LIN {X 0,Y 573.262,Z 487.391,A -85,B 0,C 180,E1 -2001.147,E2 -2001.147} C_VEL
LIN {X 0,Y 573.234,Z 487.393,A -85,B 0,C 180,E1 -2003.866,E2 -2003.866} C_VEL
LIN {X 0,Y 573.24,Z 487.393,A -85,B 0,C 180,E1 -2006.493,E2 -2006.493} C_VEL
LIN {X 0,Y 573.269,Z 487.389,A -85,B 0,C 180,E1 -2009.366,E2 -2009.366} C_VEL
LIN {X 0,Y 573.254,Z 487.391,A -85,B 0,C 180,E1 -2012.228,E2 -2012.228} C_VEL
LIN {X 0,Y 573.245,Z 487.394,A -85,B 0,C 180,E1 -2014.772,E2 -2014.772} C_VEL
LIN {X 0,Y 573.257,Z 487.391,A -85,B 0,C 180,E1 -2017.166,E2 -2017.166} C_VEL
LIN {X 0,Y 573.251,Z 487.39,A -85,B 0,C 180,E1 -2019.607,E2 -2019.607} C_VEL
LIN {X 0,Y 573.244,Z 487.391,A -85,B 0,C 180,E1 -2022.642,E2 -2022.642} C_VEL
LIN {X 0,Y 573.243,Z 487.392,A -85,B 0,C 180,E1 -2025.667,E2 -2025.667} C_VEL
LIN {X 0,Y 573.245,Z 487.392,A -85,B 0,C 180,E1 -2028.544,E2 -2028.544} C_VEL
LIN {X 0,Y 573.25,Z 487.391,A -85,B 0,C 180,E1 -2031.299,E2 -2031.299} C_VEL
LIN {X 0,Y 573.218,Z 487.395,A -85,B 0,C 180,E1 -2034.018,E2 -2034.018} C_VEL
LIN {X 0,Y 573.275,Z 487.389,A -85,B 0,C 180,E1 -2036.518,E2 -2036.518} C_VEL
LIN {X 0,Y 573.235,Z 487.396,A -85,B 0,C 180,E1 -2039.118,E2 -2039.118} C_VEL
LIN {X 0,Y 573.256,Z 487.393,A -85,B 0,C 180,E1 -2041.971,E2 -2041.971} C_VEL
LIN {X 0,Y 573.26,Z 487.394,A -85,B 0,C 180,E1 -2044.59,E2 -2044.59} C_VEL
LIN {X 0,Y 573.269,Z 487.559,A -85,B 0,C 180,E1 -2046.04,E2 -2046.04} C_VEL
LIN {X 0,Y 573.243,Z 493.535,A -85,B 0,C 180,E1 -2049.173,E2 -2049.173} C_VEL
LIN {X 0,Y 573.218,Z 499.051,A -85,B 0,C 180,E1 -2052.15,E2 -2052.15} C_VEL
LIN {X 0,Y 573.185,Z 504.475,A -85,B 0,C 180,E1 -2055.078,E2 -2055.078} C_VEL
LIN {X 0,Y 573.138,Z 509.987,A -85,B 0,C 180,E1 -2057.967,E2 -2057.967} C_VEL
LIN {X 0,Y 573.109,Z 515.58,A -85,B 0,C 180,E1 -2060.826,E2 -2060.826} C_VEL
LIN {X 0,Y 573.103,Z 521.654,A -85,B 0,C 180,E1 -2063.862,E2 -2063.862} C_VEL
LIN {X 0,Y 575.503,Z 530.402,A -85,B 0,C 180,E1 -2064.085,E2 -2064.085} C_VEL
LIN {X 0,Y 575.411,Z 546.369,A -85,B 0,C 180,E1 -2064.392,E2 -2064.392} C_VEL
LIN {X 0,Y 575.192,Z 562.192,A -85,B 0,C 180,E1 -2064.829,E2 -2064.829} C_VEL
LIN {X 0,Y 574.934,Z 579.816,A -85,B 0,C 180,E1 -2065.486,E2 -2065.486} C_VEL
LIN {X 0,Y 574.704,Z 595.268,A -85,B 0,C 180,E1 -2066.231,E2 -2066.231} C_VEL
LIN {X 0,Y 574.427,Z 610.317,A -85,B 0,C 180,E1 -2067.106,E2 -2067.106} C_VEL
LIN {X 0,Y 574.123,Z 625.23,A -85,B 0,C 180,E1 -2068.158,E2 -2068.158} C_VEL
LIN {X 0,Y 573.909,Z 636.875,A -85,B 0,C 180,E1 -2069.122,E2 -2069.122} C_VEL
LIN {X 0,Y 573.659,Z 649.57,A -85,B 0,C 180,E1 -2070.35,E2 -2070.35} C_VEL
LIN {X 0,Y 573.432,Z 661.888,A -85,B 0,C 180,E1 -2071.755,E2 -2071.755} C_VEL
LIN {X 0,Y 573.288,Z 672.217,A -85,B 0,C 180,E1 -2073.162,E2 -2073.162} C_VEL
LIN {X 0,Y 573.154,Z 680.969,A -85,B 0,C 180,E1 -2074.571,E2 -2074.571} C_VEL
LIN {X 0,Y 573.114,Z 688.382,A -85,B 0,C 180,E1 -2075.982,E2 -2075.982} C_VEL
LIN {X 0,Y 573.045,Z 694.49,A -85,B 0,C 180,E1 -2077.398,E2 -2077.398} C_VEL
LIN {X 0,Y 572.999,Z 699.458,A -85,B 0,C 180,E1 -2078.818,E2 -2078.818} C_VEL
LIN {X 0,Y 572.983,Z 704.181,A -85,B 0,C 180,E1 -2080.601,E2 -2080.601} C_VEL
LIN {X 0,Y 572.944,Z 706.767,A -85,B 0,C 180,E1 -2082.035,E2 -2082.035} C_VEL
LIN {X 0,Y 572.964,Z 708.381,A -85,B 0,C 180,E1 -2083.476,E2 -2083.476} C_VEL
LIN {X 0,Y 572.898,Z 708.98,A -85,B 0,C 180,E1 -2084.928,E2 -2084.928} C_VEL
LIN {X 0,Y 572.924,Z 708.532,A -85,B 0,C 180,E1 -2086.387,E2 -2086.387} C_VEL
LIN {X 0,Y 572.941,Z 707.077,A -85,B 0,C 180,E1 -2087.857,E2 -2087.857} C_VEL
LIN {X 0,Y 572.949,Z 704.49,A -85,B 0,C 180,E1 -2089.34,E2 -2089.34} C_VEL
LIN {X 0,Y 572.987,Z 700.765,A -85,B 0,C 180,E1 -2090.835,E2 -2090.835} C_VEL
LIN {X 0,Y 573.004,Z 695.804,A -85,B 0,C 180,E1 -2092.346,E2 -2092.346} C_VEL
LIN {X 0,Y 573.079,Z 689.462,A -85,B 0,C 180,E1 -2093.871,E2 -2093.871} C_VEL
LIN {X 0,Y 573.146,Z 681.566,A -85,B 0,C 180,E1 -2095.414,E2 -2095.414} C_VEL
LIN {X 0,Y 573.244,Z 673.765,A -85,B 0,C 180,E1 -2096.698,E2 -2096.698} C_VEL
LIN {X 0,Y 573.381,Z 664.059,A -85,B 0,C 180,E1 -2098.052,E2 -2098.052} C_VEL
LIN {X 0,Y 573.575,Z 653.23,A -85,B 0,C 180,E1 -2099.347,E2 -2099.347} C_VEL
LIN {X 0,Y 573.859,Z 640.374,A -85,B 0,C 180,E1 -2100.648,E2 -2100.648} C_VEL
LIN {X 0,Y 574.064,Z 627.395,A -85,B 0,C 180,E1 -2101.763,E2 -2101.763} C_VEL
LIN {X 0,Y 574.346,Z 613.444,A -85,B 0,C 180,E1 -2102.782,E2 -2102.782} C_VEL
LIN {X 0,Y 574.63,Z 597.773,A -85,B 0,C 180,E1 -2103.728,E2 -2103.728} C_VEL
LIN {X 0,Y 574.874,Z 583.699,A -85,B 0,C 180,E1 -2104.43,E2 -2104.43} C_VEL
LIN {X 0,Y 575.109,Z 568.288,A -85,B 0,C 180,E1 -2105.053,E2 -2105.053} C_VEL
LIN {X 0,Y 575.366,Z 551.011,A -85,B 0,C 180,E1 -2105.584,E2 -2105.584} C_VEL
LIN {X 0,Y 575.527,Z 534.59,A -85,B 0,C 180,E1 -2105.936,E2 -2105.936} C_VEL
LIN {X 0,Y 575.398,Z 530.006,A -85,B 0,C 180,E1 -2106.015,E2 -2106.015} C_VEL
LIN {X 0,Y 573.07,Z 521.633,A -85,B 0,C 180,E1 -2106.24,E2 -2106.24} C_VEL
LIN {X 0,Y 573.071,Z 516.673,A -85,B 0,C 180,E1 -2108.714,E2 -2108.714} C_VEL
LIN {X 0,Y 573.119,Z 511.04,A -85,B 0,C 180,E1 -2111.58,E2 -2111.58} C_VEL
LIN {X 0,Y 573.168,Z 505.123,A -85,B 0,C 180,E1 -2114.669,E2 -2114.669} C_VEL
LIN {X 0,Y 573.2,Z 500.111,A -85,B 0,C 180,E1 -2117.361,E2 -2117.361} C_VEL
LIN {X 0,Y 573.222,Z 494.449,A -85,B 0,C 180,E1 -2120.39,E2 -2120.39} C_VEL
LIN {X 0,Y 573.209,Z 489.4,A -85,B 0,C 180,E1 -2123.074,E2 -2123.074} C_VEL
LIN {X 0,Y 573.254,Z 487.395,A -85,B 0,C 180,E1 -2124.076,E2 -2124.076} C_VEL
LIN {X 0,Y 573.278,Z 487.391,A -85,B 0,C 180,E1 -2126.518,E2 -2126.518} C_VEL
LIN {X 0,Y 573.237,Z 487.395,A -85,B 0,C 180,E1 -2129.114,E2 -2129.114} C_VEL
LIN {X 0,Y 573.257,Z 487.393,A -85,B 0,C 180,E1 -2131.967,E2 -2131.967} C_VEL
LIN {X 0,Y 573.252,Z 487.393,A -85,B 0,C 180,E1 -2134.589,E2 -2134.589} C_VEL
LIN {X 0,Y 573.255,Z 487.39,A -85,B 0,C 180,E1 -2136.901,E2 -2136.901} C_VEL
LIN {X 0,Y 573.247,Z 487.392,A -85,B 0,C 180,E1 -2139.923,E2 -2139.923} C_VEL
LIN {X 0,Y 573.255,Z 487.395,A -85,B 0,C 180,E1 -2142.987,E2 -2142.987} C_VEL
LIN {X 0,Y 573.264,Z 487.392,A -85,B 0,C 180,E1 -2145.806,E2 -2145.806} C_VEL
LIN {X 0,Y 573.273,Z 487.389,A -85,B 0,C 180,E1 -2148.733,E2 -2148.733} C_VEL
LIN {X 0,Y 573.3,Z 487.385,A -85,B 0,C 180,E1 -2151.54,E2 -2151.54} C_VEL
LIN {X 0,Y 573.295,Z 487.385,A -85,B 0,C 180,E1 -2154.372,E2 -2154.372} C_VEL
LIN {X 0,Y 573.31,Z 487.387,A -85,B 0,C 180,E1 -2157.892,E2 -2157.892} C_VEL
LIN {X 0,Y 573.331,Z 487.385,A -85,B 0,C 180,E1 -2160.702,E2 -2160.702} C_VEL
LIN {X 0,Y 573.234,Z 487.396,A -85,B 0,C 180,E1 -2163.514,E2 -2163.514} C_VEL
LIN {X 0,Y 573.284,Z 487.385,A -85,B 0,C 180,E1 -2165.628,E2 -2165.628} C_VEL
LIN {X 0,Y 573.298,Z 487.385,A -85,B 0,C 180,E1 -2168.459,E2 -2168.459} C_VEL
LIN {X 0,Y 573.288,Z 487.388,A -85,B 0,C 180,E1 -2171.311,E2 -2171.311} C_VEL
LIN {X 0,Y 573.27,Z 487.391,A -85,B 0,C 180,E1 -2174.425,E2 -2174.425} C_VEL
LIN {X 0,Y 573.249,Z 487.387,A -85,B 0,C 180,E1 -2177.112,E2 -2177.112} C_VEL
LIN {X 0,Y 573.248,Z 487.392,A -85,B 0,C 180,E1 -2180.076,E2 -2180.076} C_VEL
LIN {X 0,Y 573.261,Z 487.388,A -85,B 0,C 180,E1 -2183.154,E2 -2183.154} C_VEL
LIN {X 0,Y 573.281,Z 487.386,A -85,B 0,C 180,E1 -2186.189,E2 -2186.189} C_VEL
LIN {X 0,Y 573.234,Z 487.393,A -85,B 0,C 180,E1 -2188.564,E2 -2188.564} C_VEL
LIN {X 0,Y 573.231,Z 487.394,A -85,B 0,C 180,E1 -2190.993,E2 -2190.993} C_VEL
LIN {X 0,Y 573.278,Z 487.389,A -85,B 0,C 180,E1 -2193.529,E2 -2193.529} C_VEL
LIN {X 0,Y 573.253,Z 487.394,A -85,B 0,C 180,E1 -2196.048,E2 -2196.048} C_VEL
LIN {X 0,Y 573.241,Z 487.396,A -85,B 0,C 180,E1 -2198.701,E2 -2198.701} C_VEL
LIN {X 0,Y 573.257,Z 487.393,A -85,B 0,C 180,E1 -2201.598,E2 -2201.598} C_VEL
LIN {X 0,Y 573.23,Z 487.397,A -85,B 0,C 180,E1 -2204.334,E2 -2204.334} C_VEL
LIN {X 0,Y 573.253,Z 487.393,A -85,B 0,C 180,E1 -2207.357,E2 -2207.357} C_VEL
LIN {X 0,Y 573.267,Z 487.459,A -85,B 0,C 180,E1 -2208.403,E2 -2208.403} C_VEL
LIN {X 0,Y 574.646,Z 493.703,A -85,B 0,C 180,E1 -2210.046,E2 -2210.046} C_VEL
LIN {X 0,Y 574.7,Z 501.177,A -85,B 0,C 180,E1 -2211.906,E2 -2211.906} C_VEL
LIN {X 0,Y 574.476,Z 511.898,A -85,B 0,C 180,E1 -2214.473,E2 -2214.473} C_VEL
LIN {X 0,Y 574.26,Z 522.796,A -85,B 0,C 180,E1 -2217.004,E2 -2217.004} C_VEL
LIN {X 0,Y 574.097,Z 535.51,A -85,B 0,C 180,E1 -2219.874,E2 -2219.874} C_VEL
LIN {X 0,Y 573.926,Z 548.224,A -85,B 0,C 180,E1 -2222.665,E2 -2222.665} C_VEL
LIN {X 0,Y 573.714,Z 560.938,A -85,B 0,C 180,E1 -2225.387,E2 -2225.387} C_VEL
LIN {X 0,Y 573.592,Z 573.652,A -85,B 0,C 180,E1 -2228.057,E2 -2228.057} C_VEL
LIN {X 0,Y 573.576,Z 577.286,A -85,B 0,C 180,E1 -2228.785,E2 -2228.785} C_VEL
LIN {X 0,Y 575.538,Z 585.817,A -85,B 0,C 180,E1 -2228.972,E2 -2228.972} C_VEL
LIN {X 0,Y 575.425,Z 602.393,A -85,B 0,C 180,E1 -2229.257,E2 -2229.257} C_VEL
LIN {X 0,Y 575.273,Z 618.484,A -85,B 0,C 180,E1 -2229.672,E2 -2229.672} C_VEL
LIN {X 0,Y 575.028,Z 635.073,A -85,B 0,C 180,E1 -2230.249,E2 -2230.249} C_VEL
LIN {X 0,Y 574.764,Z 650.013,A -85,B 0,C 180,E1 -2230.909,E2 -2230.909} C_VEL
LIN {X 0,Y 574.509,Z 665.029,A -85,B 0,C 180,E1 -2231.732,E2 -2231.732} C_VEL
LIN {X 0,Y 574.21,Z 679.457,A -85,B 0,C 180,E1 -2232.682,E2 -2232.682} C_VEL
LIN {X 0,Y 573.971,Z 692.926,A -85,B 0,C 180,E1 -2233.735,E2 -2233.735} C_VEL
LIN {X 0,Y 573.729,Z 705.738,A -85,B 0,C 180,E1 -2234.913,E2 -2234.913} C_VEL
LIN {X 0,Y 573.511,Z 717.451,A -85,B 0,C 180,E1 -2236.176,E2 -2236.176} C_VEL
LIN {X 0,Y 573.33,Z 728.738,A -85,B 0,C 180,E1 -2237.614,E2 -2237.614} C_VEL
LIN {X 0,Y 573.204,Z 738.357,A -85,B 0,C 180,E1 -2239.074,E2 -2239.074} C_VEL
LIN {X 0,Y 573.109,Z 746.053,A -85,B 0,C 180,E1 -2240.472,E2 -2240.472} C_VEL
LIN {X 0,Y 573.054,Z 752.628,A -85,B 0,C 180,E1 -2241.893,E2 -2241.893} C_VEL
LIN {X 0,Y 573.025,Z 758.391,A -85,B 0,C 180,E1 -2243.433,E2 -2243.433} C_VEL
LIN {X 0,Y 573.035,Z 761.249,A -85,B 0,C 180,E1 -2244.37,E2 -2244.37} C_VEL
LIN {X 0,Y 573.006,Z 764.636,A -85,B 0,C 180,E1 -2245.781,E2 -2245.781} C_VEL
LIN {X 0,Y 572.947,Z 767.089,A -85,B 0,C 180,E1 -2247.188,E2 -2247.188} C_VEL
LIN {X 0,Y 572.943,Z 768.479,A -85,B 0,C 180,E1 -2248.595,E2 -2248.595} C_VEL
LIN {X 0,Y 572.933,Z 769,A -85,B 0,C 180,E1 -2250.001,E2 -2250.001} C_VEL
LIN {X 0,Y 572.943,Z 768.478,A -85,B 0,C 180,E1 -2251.407,E2 -2251.407} C_VEL
LIN {X 0,Y 572.947,Z 767.086,A -85,B 0,C 180,E1 -2252.813,E2 -2252.813} C_VEL
LIN {X 0,Y 573.006,Z 764.633,A -85,B 0,C 180,E1 -2254.221,E2 -2254.221} C_VEL
LIN {X 0,Y 573.012,Z 760.184,A -85,B 0,C 180,E1 -2255.985,E2 -2255.985} C_VEL
LIN {X 0,Y 573.043,Z 755.466,A -85,B 0,C 180,E1 -2257.4,E2 -2257.4} C_VEL
LIN {X 0,Y 573.092,Z 747.854,A -85,B 0,C 180,E1 -2259.174,E2 -2259.174} C_VEL
LIN {X 0,Y 573.15,Z 740.257,A -85,B 0,C 180,E1 -2260.599,E2 -2260.599} C_VEL
LIN {X 0,Y 573.304,Z 731.205,A -85,B 0,C 180,E1 -2262.029,E2 -2262.029} C_VEL
LIN {X 0,Y 573.442,Z 720.418,A -85,B 0,C 180,E1 -2263.466,E2 -2263.466} C_VEL
LIN {X 0,Y 573.658,Z 709.292,A -85,B 0,C 180,E1 -2264.726,E2 -2264.726} C_VEL
LIN {X 0,Y 573.902,Z 697.137,A -85,B 0,C 180,E1 -2265.903,E2 -2265.903} C_VEL
LIN {X 0,Y 574.132,Z 683.875,A -85,B 0,C 180,E1 -2266.994,E2 -2266.994} C_VEL
LIN {X 0,Y 574.431,Z 669.425,A -85,B 0,C 180,E1 -2267.995,E2 -2267.995} C_VEL
LIN {X 0,Y 574.662,Z 655.255,A -85,B 0,C 180,E1 -2268.818,E2 -2268.818} C_VEL
LIN {X 0,Y 574.935,Z 640.706,A -85,B 0,C 180,E1 -2269.521,E2 -2269.521} C_VEL
LIN {X 0,Y 575.198,Z 624.331,A -85,B 0,C 180,E1 -2270.146,E2 -2270.146} C_VEL
LIN {X 0,Y 575.387,Z 608.329,A -85,B 0,C 180,E1 -2270.606,E2 -2270.606} C_VEL
LIN {X 0,Y 575.518,Z 591.668,A -85,B 0,C 180,E1 -2270.94,E2 -2270.94} C_VEL
LIN {X 0,Y 575.396,Z 584.289,A -85,B 0,C 180,E1 -2271.053,E2 -2271.053} C_VEL
LIN {X 0,Y 573.548,Z 577.09,A -85,B 0,C 180,E1 -2271.23,E2 -2271.23} C_VEL
LIN {X 0,Y 573.695,Z 562.746,A -85,B 0,C 180,E1 -2274.23,E2 -2274.23} C_VEL
LIN {X 0,Y 573.889,Z 550.032,A -85,B 0,C 180,E1 -2276.944,E2 -2276.944} C_VEL
LIN {X 0,Y 574.052,Z 536.852,A -85,B 0,C 180,E1 -2279.829,E2 -2279.829} C_VEL
LIN {X 0,Y 574.247,Z 524.604,A -85,B 0,C 180,E1 -2282.582,E2 -2282.582} C_VEL
LIN {X 0,Y 574.398,Z 513.707,A -85,B 0,C 180,E1 -2285.105,E2 -2285.105} C_VEL
LIN {X 0,Y 574.654,Z 502.809,A -85,B 0,C 180,E1 -2287.698,E2 -2287.698} C_VEL
LIN {X 0,Y 574.733,Z 495.035,A -85,B 0,C 180,E1 -2289.612,E2 -2289.612} C_VEL
LIN {X 0,Y 573.722,Z 489.451,A -85,B 0,C 180,E1 -2291.076,E2 -2291.076} C_VEL
LIN {X 0,Y 573.26,Z 487.39,A -85,B 0,C 180,E1 -2291.539,E2 -2291.539} C_VEL
LIN {X 0,Y 573.241,Z 487.392,A -85,B 0,C 180,E1 -2294.333,E2 -2294.333} C_VEL
LIN {X 0,Y 573.244,Z 487.389,A -85,B 0,C 180,E1 -2297.358,E2 -2297.358} C_VEL
LIN {X 0,Y 573.249,Z 487.394,A -85,B 0,C 180,E1 -2300.393,E2 -2300.393} C_VEL
LIN {X 0,Y 573.253,Z 487.388,A -85,B 0,C 180,E1 -2303.078,E2 -2303.078} C_VEL
LIN {X 0,Y 573.272,Z 487.385,A -85,B 0,C 180,E1 -2305.672,E2 -2305.672} C_VEL
LIN {X 0,Y 573.242,Z 487.396,A -85,B 0,C 180,E1 -2308.185,E2 -2308.185} C_VEL
LIN {X 0,Y 573.267,Z 487.388,A -85,B 0,C 180,E1 -2310.635,E2 -2310.635} C_VEL
LIN {X 0,Y 573.252,Z 487.387,A -85,B 0,C 180,E1 -2313.024,E2 -2313.024} C_VEL
LIN {X 0,Y 573.277,Z 487.386,A -85,B 0,C 180,E1 -2315.366,E2 -2315.366} C_VEL
LIN {X 0,Y 573.231,Z 487.393,A -85,B 0,C 180,E1 -2318.42,E2 -2318.42} C_VEL
LIN {X 0,Y 573.265,Z 487.387,A -85,B 0,C 180,E1 -2318.952,E2 -2318.952} C_VEL
LIN {X 0,Y 575.047,Z 492.214,A -85,B 0,C 180,E1 -2319.094,E2 -2319.094} C_VEL
LIN {X 0,Y 575.537,Z 494.378,A -85,B 0,C 180,E1 -2319.147,E2 -2319.147} C_VEL
LIN {X 0,Y 575.338,Z 511.225,A -85,B 0,C 180,E1 -2319.51,E2 -2319.51} C_VEL
LIN {X 0,Y 575.13,Z 527.051,A -85,B 0,C 180,E1 -2319.992,E2 -2319.992} C_VEL
LIN {X 0,Y 574.918,Z 543.212,A -85,B 0,C 180,E1 -2320.637,E2 -2320.637} C_VEL
LIN {X 0,Y 574.637,Z 557.901,A -85,B 0,C 180,E1 -2321.367,E2 -2321.367} C_VEL
LIN {X 0,Y 574.38,Z 572.82,A -85,B 0,C 180,E1 -2322.27,E2 -2322.27} C_VEL
LIN {X 0,Y 574.107,Z 586.828,A -85,B 0,C 180,E1 -2323.281,E2 -2323.281} C_VEL
LIN {X 0,Y 573.826,Z 599.609,A -85,B 0,C 180,E1 -2324.369,E2 -2324.369} C_VEL
LIN {X 0,Y 573.632,Z 611.874,A -85,B 0,C 180,E1 -2325.594,E2 -2325.594} C_VEL
LIN {X 0,Y 573.419,Z 622.99,A -85,B 0,C 180,E1 -2326.895,E2 -2326.895} C_VEL
LIN {X 0,Y 573.288,Z 633.371,A -85,B 0,C 180,E1 -2328.33,E2 -2328.33} C_VEL
LIN {X 0,Y 573.169,Z 642.045,A -85,B 0,C 180,E1 -2329.759,E2 -2329.759} C_VEL
LIN {X 0,Y 573.086,Z 649.296,A -85,B 0,C 180,E1 -2331.183,E2 -2331.183} C_VEL
LIN {X 0,Y 573.044,Z 655.298,A -85,B 0,C 180,E1 -2332.601,E2 -2332.601} C_VEL
LIN {X 0,Y 573.014,Z 660.066,A -85,B 0,C 180,E1 -2334.016,E2 -2334.016} C_VEL
LIN {X 0,Y 573.005,Z 664.546,A -85,B 0,C 180,E1 -2335.78,E2 -2335.78} C_VEL
LIN {X 0,Y 572.954,Z 667.024,A -85,B 0,C 180,E1 -2337.188,E2 -2337.188} C_VEL
LIN {X 0,Y 572.939,Z 668.459,A -85,B 0,C 180,E1 -2338.595,E2 -2338.595} C_VEL
LIN {X 0,Y 572.935,Z 668.996,A -85,B 0,C 180,E1 -2340,E2 -2340} C_VEL
LIN {X 0,Y 572.939,Z 668.518,A -85,B 0,C 180,E1 -2341.406,E2 -2341.406} C_VEL
LIN {X 0,Y 572.954,Z 667.141,A -85,B 0,C 180,E1 -2342.813,E2 -2342.813} C_VEL
LIN {X 0,Y 573.006,Z 664.733,A -85,B 0,C 180,E1 -2344.221,E2 -2344.221} C_VEL
LIN {X 0,Y 573.017,Z 660.331,A -85,B 0,C 180,E1 -2345.984,E2 -2345.984} C_VEL
LIN {X 0,Y 573.044,Z 655.624,A -85,B 0,C 180,E1 -2347.399,E2 -2347.399} C_VEL
LIN {X 0,Y 573.082,Z 649.694,A -85,B 0,C 180,E1 -2348.818,E2 -2348.818} C_VEL
LIN {X 0,Y 573.186,Z 641.542,A -85,B 0,C 180,E1 -2350.42,E2 -2350.42} C_VEL
LIN {X 0,Y 573.271,Z 632.765,A -85,B 0,C 180,E1 -2351.85,E2 -2351.85} C_VEL
LIN {X 0,Y 573.437,Z 622.274,A -85,B 0,C 180,E1 -2353.286,E2 -2353.286} C_VEL
LIN {X 0,Y 573.638,Z 610.405,A -85,B 0,C 180,E1 -2354.655,E2 -2354.655} C_VEL
LIN {X 0,Y 573.86,Z 598.613,A -85,B 0,C 180,E1 -2355.813,E2 -2355.813} C_VEL
LIN {X 0,Y 574.115,Z 585.624,A -85,B 0,C 180,E1 -2356.902,E2 -2356.902} C_VEL
LIN {X 0,Y 574.378,Z 571.555,A -85,B 0,C 180,E1 -2357.904,E2 -2357.904} C_VEL
LIN {X 0,Y 574.652,Z 557.869,A -85,B 0,C 180,E1 -2358.726,E2 -2358.726} C_VEL
LIN {X 0,Y 574.939,Z 541.855,A -85,B 0,C 180,E1 -2359.515,E2 -2359.515} C_VEL
LIN {X 0,Y 574.989,Z 538.259,A -85,B 0,C 180,E1 -2359.667,E2 -2359.667} C_VEL
LIN {X 0,Y 574.341,Z 534.687,A -85,B 0,C 180,E1 -2359.839,E2 -2359.839} C_VEL
LIN {X 0,Y 569.101,Z 523.749,A -85,B 0,C 180,E1 -2360.438,E2 -2360.438} C_VEL
LIN {X 0,Y 568.59,Z 520.064,A -85,B 0,C 180,E1 -2360.573,E2 -2360.573} C_VEL
LIN {X 0,Y 568.788,Z 505.313,A -85,B 0,C 180,E1 -2360.974,E2 -2360.974} C_VEL
LIN {X 0,Y 568.718,Z 494.777,A -85,B 0,C 180,E1 -2361.195,E2 -2361.195} C_VEL
LIN {X 0,Y 566.315,Z 488.81,A -85,B 0,C 180,E1 -2361.387,E2 -2361.387} C_VEL
LIN {X 0,Y 566.221,Z 488.269,A -85,B 0,C 180,E1 -2361.423,E2 -2361.423} C_VEL
LIN {X 0,Y 566.201,Z 488.27,A -85,B 0,C 180,E1 -2364.181,E2 -2364.181} C_VEL
LIN {X 0,Y 566.211,Z 488.268,A -85,B 0,C 180,E1 -2366.659,E2 -2366.659} C_VEL
LIN {X 0,Y 566.196,Z 488.274,A -85,B 0,C 180,E1 -2368.954,E2 -2368.954} C_VEL
LIN {X 0,Y 566.196,Z 488.271,A -85,B 0,C 180,E1 -2371.422,E2 -2371.422} C_VEL
LIN {X 0,Y 566.215,Z 488.267,A -85,B 0,C 180,E1 -2373.956,E2 -2373.956} C_VEL
LIN {X 0,Y 566.219,Z 488.266,A -85,B 0,C 180,E1 -2376.569,E2 -2376.569} C_VEL
LIN {X 0,Y 566.226,Z 488.265,A -85,B 0,C 180,E1 -2379.687,E2 -2379.687} C_VEL
LIN {X 0,Y 566.206,Z 488.27,A -85,B 0,C 180,E1 -2382.917,E2 -2382.917} C_VEL
LIN {X 0,Y 566.207,Z 488.273,A -85,B 0,C 180,E1 -2386.048,E2 -2386.048} C_VEL
LIN {X 0,Y 566.214,Z 488.271,A -85,B 0,C 180,E1 -2388.864,E2 -2388.864} C_VEL
LIN {X 0,Y 566.192,Z 488.273,A -85,B 0,C 180,E1 -2391.637,E2 -2391.637} C_VEL
LIN {X 0,Y 566.168,Z 488.275,A -85,B 0,C 180,E1 -2394.308,E2 -2394.308} C_VEL
LIN {X 0,Y 566.226,Z 488.266,A -85,B 0,C 180,E1 -2396.898,E2 -2396.898} C_VEL
LIN {X 0,Y 566.187,Z 488.272,A -85,B 0,C 180,E1 -2399.407,E2 -2399.407} C_VEL
LIN {X 0,Y 566.218,Z 488.271,A -85,B 0,C 180,E1 -2401.857,E2 -2401.857} C_VEL
LIN {X 0,Y 566.22,Z 488.268,A -85,B 0,C 180,E1 -2404.251,E2 -2404.251} C_VEL
LIN {X 0,Y 566.233,Z 488.393,A -85,B 0,C 180,E1 -2406.015,E2 -2406.015} C_VEL
LIN {X 0,Y 566.204,Z 493.917,A -85,B 0,C 180,E1 -2408.902,E2 -2408.902} C_VEL
LIN {X 0,Y 566.172,Z 498.111,A -85,B 0,C 180,E1 -2411.171,E2 -2411.171} C_VEL
LIN {X 0,Y 566.115,Z 503.525,A -85,B 0,C 180,E1 -2414.15,E2 -2414.15} C_VEL
LIN {X 0,Y 566.106,Z 507.629,A -85,B 0,C 180,E1 -2416.356,E2 -2416.356} C_VEL
LIN {X 0,Y 566.061,Z 513.177,A -85,B 0,C 180,E1 -2419.266,E2 -2419.266} C_VEL
LIN {X 0,Y 566.038,Z 518.808,A -85,B 0,C 180,E1 -2422.149,E2 -2422.149} C_VEL
LIN {X 0,Y 566.046,Z 521.652,A -85,B 0,C 180,E1 -2423.583,E2 -2423.583} C_VEL
LIN {X 0,Y 568.894,Z 532.268,A -85,B 0,C 180,E1 -2423.861,E2 -2423.861} C_VEL
LIN {X 0,Y 568.745,Z 548.595,A -85,B 0,C 180,E1 -2424.193,E2 -2424.193} C_VEL
LIN {X 0,Y 568.475,Z 566.381,A -85,B 0,C 180,E1 -2424.724,E2 -2424.724} C_VEL
LIN {X 0,Y 568.181,Z 581,A -85,B 0,C 180,E1 -2425.299,E2 -2425.299} C_VEL
LIN {X 0,Y 567.92,Z 595.456,A -85,B 0,C 180,E1 -2426.008,E2 -2426.008} C_VEL
LIN {X 0,Y 567.595,Z 610.488,A -85,B 0,C 180,E1 -2426.894,E2 -2426.894} C_VEL
LIN {X 0,Y 567.255,Z 625.366,A -85,B 0,C 180,E1 -2427.958,E2 -2427.958} C_VEL
LIN {X 0,Y 566.997,Z 636.987,A -85,B 0,C 180,E1 -2428.934,E2 -2428.934} C_VEL
LIN {X 0,Y 566.688,Z 649.676,A -85,B 0,C 180,E1 -2430.177,E2 -2430.177} C_VEL
LIN {X 0,Y 566.41,Z 661.983,A -85,B 0,C 180,E1 -2431.599,E2 -2431.599} C_VEL
LIN {X 0,Y 566.251,Z 672.285,A -85,B 0,C 180,E1 -2433.023,E2 -2433.023} C_VEL
LIN {X 0,Y 566.117,Z 681.027,A -85,B 0,C 180,E1 -2434.449,E2 -2434.449} C_VEL
LIN {X 0,Y 566.029,Z 689.237,A -85,B 0,C 180,E1 -2436.057,E2 -2436.057} C_VEL
LIN {X 0,Y 565.972,Z 695.228,A -85,B 0,C 180,E1 -2437.491,E2 -2437.491} C_VEL
LIN {X 0,Y 565.895,Z 700.022,A -85,B 0,C 180,E1 -2438.93,E2 -2438.93} C_VEL
LIN {X 0,Y 565.9,Z 702.958,A -85,B 0,C 180,E1 -2440.012,E2 -2440.012} C_VEL
LIN {X 0,Y 565.873,Z 705.93,A -85,B 0,C 180,E1 -2441.461,E2 -2441.461} C_VEL
LIN {X 0,Y 565.838,Z 707.906,A -85,B 0,C 180,E1 -2442.918,E2 -2442.918} C_VEL
LIN {X 0,Y 565.84,Z 708.856,A -85,B 0,C 180,E1 -2444.382,E2 -2444.382} C_VEL
LIN {X 0,Y 565.804,Z 708.809,A -85,B 0,C 180,E1 -2445.858,E2 -2445.858} C_VEL
LIN {X 0,Y 565.83,Z 707.72,A -85,B 0,C 180,E1 -2447.342,E2 -2447.342} C_VEL
LIN {X 0,Y 565.85,Z 705.599,A -85,B 0,C 180,E1 -2448.839,E2 -2448.839} C_VEL
LIN {X 0,Y 565.89,Z 702.287,A -85,B 0,C 180,E1 -2450.348,E2 -2450.348} C_VEL
LIN {X 0,Y 565.931,Z 697.776,A -85,B 0,C 180,E1 -2451.872,E2 -2451.872} C_VEL
LIN {X 0,Y 565.977,Z 691.966,A -85,B 0,C 180,E1 -2453.412,E2 -2453.412} C_VEL
LIN {X 0,Y 566.035,Z 686.622,A -85,B 0,C 180,E1 -2454.578,E2 -2454.578} C_VEL
LIN {X 0,Y 566.174,Z 678.134,A -85,B 0,C 180,E1 -2456.145,E2 -2456.145} C_VEL
LIN {X 0,Y 566.315,Z 667.674,A -85,B 0,C 180,E1 -2457.733,E2 -2457.733} C_VEL
LIN {X 0,Y 566.485,Z 658.349,A -85,B 0,C 180,E1 -2458.936,E2 -2458.936} C_VEL
LIN {X 0,Y 566.726,Z 647.425,A -85,B 0,C 180,E1 -2460.147,E2 -2460.147} C_VEL
LIN {X 0,Y 566.995,Z 636.403,A -85,B 0,C 180,E1 -2461.21,E2 -2461.21} C_VEL
LIN {X 0,Y 567.279,Z 622.959,A -85,B 0,C 180,E1 -2462.324,E2 -2462.324} C_VEL
LIN {X 0,Y 567.63,Z 608.469,A -85,B 0,C 180,E1 -2463.326,E2 -2463.326} C_VEL
LIN {X 0,Y 567.889,Z 595.643,A -85,B 0,C 180,E1 -2464.073,E2 -2464.073} C_VEL
LIN {X 0,Y 568.171,Z 581.485,A -85,B 0,C 180,E1 -2464.769,E2 -2464.769} C_VEL
LIN {X 0,Y 568.438,Z 566.657,A -85,B 0,C 180,E1 -2465.358,E2 -2465.358} C_VEL
LIN {X 0,Y 568.699,Z 548.636,A -85,B 0,C 180,E1 -2465.898,E2 -2465.898} C_VEL
LIN {X 0,Y 568.902,Z 532.727,A -85,B 0,C 180,E1 -2466.222,E2 -2466.222} C_VEL
LIN {X 0,Y 568.39,Z 530.003,A -85,B 0,C 180,E1 -2466.286,E2 -2466.286} C_VEL
LIN {X 0,Y 565.989,Z 521.644,A -85,B 0,C 180,E1 -2466.513,E2 -2466.513} C_VEL
LIN {X 0,Y 565.999,Z 516.161,A -85,B 0,C 180,E1 -2469.29,E2 -2469.29} C_VEL
LIN {X 0,Y 566.062,Z 510.729,A -85,B 0,C 180,E1 -2472.099,E2 -2472.099} C_VEL
LIN {X 0,Y 566.126,Z 505.189,A -85,B 0,C 180,E1 -2475.039,E2 -2475.039} C_VEL
LIN {X 0,Y 566.137,Z 499.958,A -85,B 0,C 180,E1 -2477.905,E2 -2477.905} C_VEL
LIN {X 0,Y 566.172,Z 494.608,A -85,B 0,C 180,E1 -2480.722,E2 -2480.722} C_VEL
LIN {X 0,Y 566.155,Z 489.489,A -85,B 0,C 180,E1 -2483.426,E2 -2483.426} C_VEL
LIN {X 0,Y 566.204,Z 488.273,A -85,B 0,C 180,E1 -2484.048,E2 -2484.048} C_VEL
LIN {X 0,Y 566.222,Z 488.271,A -85,B 0,C 180,E1 -2486.898,E2 -2486.898} C_VEL
LIN {X 0,Y 566.187,Z 488.276,A -85,B 0,C 180,E1 -2489.407,E2 -2489.407} C_VEL
LIN {X 0,Y 566.22,Z 488.269,A -85,B 0,C 180,E1 -2491.857,E2 -2491.857} C_VEL
LIN {X 0,Y 566.22,Z 488.267,A -85,B 0,C 180,E1 -2494.251,E2 -2494.251} C_VEL
LIN {X 0,Y 566.226,Z 488.266,A -85,B 0,C 180,E1 -2496.702,E2 -2496.702} C_VEL
LIN {X 0,Y 566.21,Z 488.268,A -85,B 0,C 180,E1 -2499.662,E2 -2499.662} C_VEL
LIN {X 0,Y 566.197,Z 488.271,A -85,B 0,C 180,E1 -2502.668,E2 -2502.668} C_VEL
LIN {X 0,Y 566.225,Z 488.27,A -85,B 0,C 180,E1 -2505.626,E2 -2505.626} C_VEL
LIN {X 0,Y 566.265,Z 488.262,A -85,B 0,C 180,E1 -2508.653,E2 -2508.653} C_VEL
LIN {X 0,Y 566.242,Z 488.264,A -85,B 0,C 180,E1 -2511.434,E2 -2511.434} C_VEL
LIN {X 0,Y 566.263,Z 488.261,A -85,B 0,C 180,E1 -2514.301,E2 -2514.301} C_VEL
LIN {X 0,Y 566.28,Z 488.263,A -85,B 0,C 180,E1 -2517.866,E2 -2517.866} C_VEL
LIN {X 0,Y 566.3,Z 488.26,A -85,B 0,C 180,E1 -2520.711,E2 -2520.711} C_VEL
LIN {X 0,Y 566.271,Z 488.26,A -85,B 0,C 180,E1 -2522.845,E2 -2522.845} C_VEL
LIN {X 0,Y 566.252,Z 488.261,A -85,B 0,C 180,E1 -2525.698,E2 -2525.698} C_VEL
LIN {X 0,Y 566.239,Z 488.265,A -85,B 0,C 180,E1 -2528.565,E2 -2528.565} C_VEL
LIN {X 0,Y 566.24,Z 488.267,A -85,B 0,C 180,E1 -2531.454,E2 -2531.454} C_VEL
LIN {X 0,Y 566.223,Z 488.268,A -85,B 0,C 180,E1 -2534.507,E2 -2534.507} C_VEL
LIN {X 0,Y 566.194,Z 488.263,A -85,B 0,C 180,E1 -2537.332,E2 -2537.332} C_VEL
LIN {X 0,Y 566.21,Z 488.267,A -85,B 0,C 180,E1 -2540.337,E2 -2540.337} C_VEL
LIN {X 0,Y 566.22,Z 488.265,A -85,B 0,C 180,E1 -2543.402,E2 -2543.402} C_VEL
LIN {X 0,Y 566.218,Z 488.264,A -85,B 0,C 180,E1 -2545.748,E2 -2545.748} C_VEL
LIN {X 0,Y 566.198,Z 488.27,A -85,B 0,C 180,E1 -2548.204,E2 -2548.204} C_VEL
LIN {X 0,Y 566.185,Z 488.275,A -85,B 0,C 180,E1 -2550.592,E2 -2550.592} C_VEL
LIN {X 0,Y 566.219,Z 488.269,A -85,B 0,C 180,E1 -2553.102,E2 -2553.102} C_VEL
LIN {X 0,Y 566.204,Z 488.269,A -85,B 0,C 180,E1 -2555.689,E2 -2555.689} C_VEL
LIN {X 0,Y 566.208,Z 488.271,A -85,B 0,C 180,E1 -2558.56,E2 -2558.56} C_VEL
LIN {X 0,Y 566.213,Z 488.269,A -85,B 0,C 180,E1 -2561.136,E2 -2561.136} C_VEL
LIN {X 0,Y 566.191,Z 488.274,A -85,B 0,C 180,E1 -2564.036,E2 -2564.036} C_VEL
LIN {X 0,Y 566.206,Z 488.272,A -85,B 0,C 180,E1 -2567.082,E2 -2567.082} C_VEL
LIN {X 0,Y 566.264,Z 488.36,A -85,B 0,C 180,E1 -2568.096,E2 -2568.096} C_VEL
LIN {X 0,Y 567.902,Z 496.189,A -85,B 0,C 180,E1 -2570.109,E2 -2570.109} C_VEL
LIN {X 0,Y 567.836,Z 505.294,A -85,B 0,C 180,E1 -2572.383,E2 -2572.383} C_VEL
LIN {X 0,Y 567.563,Z 517.347,A -85,B 0,C 180,E1 -2575.279,E2 -2575.279} C_VEL
LIN {X 0,Y 567.305,Z 530.061,A -85,B 0,C 180,E1 -2578.232,E2 -2578.232} C_VEL
LIN {X 0,Y 567.06,Z 542.775,A -85,B 0,C 180,E1 -2581.096,E2 -2581.096} C_VEL
LIN {X 0,Y 566.876,Z 553.673,A -85,B 0,C 180,E1 -2583.493,E2 -2583.493} C_VEL
LIN {X 0,Y 566.694,Z 566.388,A -85,B 0,C 180,E1 -2586.232,E2 -2586.232} C_VEL
LIN {X 0,Y 566.581,Z 577.12,A -85,B 0,C 180,E1 -2588.502,E2 -2588.502} C_VEL
LIN {X 0,Y 568.936,Z 586.825,A -85,B 0,C 180,E1 -2588.73,E2 -2588.73} C_VEL
LIN {X 0,Y 568.781,Z 603.534,A -85,B 0,C 180,E1 -2589.027,E2 -2589.027} C_VEL
LIN {X 0,Y 568.583,Z 620.002,A -85,B 0,C 180,E1 -2589.469,E2 -2589.469} C_VEL
LIN {X 0,Y 568.299,Z 635.651,A -85,B 0,C 180,E1 -2590.029,E2 -2590.029} C_VEL
LIN {X 0,Y 568.027,Z 650.012,A -85,B 0,C 180,E1 -2590.673,E2 -2590.673} C_VEL
LIN {X 0,Y 567.701,Z 665.031,A -85,B 0,C 180,E1 -2591.505,E2 -2591.505} C_VEL
LIN {X 0,Y 567.386,Z 679.14,A -85,B 0,C 180,E1 -2592.444,E2 -2592.444} C_VEL
LIN {X 0,Y 567.087,Z 692.927,A -85,B 0,C 180,E1 -2593.532,E2 -2593.532} C_VEL
LIN {X 0,Y 566.828,Z 703.95,A -85,B 0,C 180,E1 -2594.54,E2 -2594.54} C_VEL
LIN {X 0,Y 566.601,Z 715.897,A -85,B 0,C 180,E1 -2595.821,E2 -2595.821} C_VEL
LIN {X 0,Y 566.364,Z 726.062,A -85,B 0,C 180,E1 -2597.094,E2 -2597.094} C_VEL
LIN {X 0,Y 566.207,Z 735.937,A -85,B 0,C 180,E1 -2598.546,E2 -2598.546} C_VEL
LIN {X 0,Y 566.084,Z 744.236,A -85,B 0,C 180,E1 -2599.991,E2 -2599.991} C_VEL
LIN {X 0,Y 566.022,Z 751.108,A -85,B 0,C 180,E1 -2601.432,E2 -2601.432} C_VEL
LIN {X 0,Y 565.965,Z 756.72,A -85,B 0,C 180,E1 -2602.868,E2 -2602.868} C_VEL
LIN {X 0,Y 565.96,Z 761.249,A -85,B 0,C 180,E1 -2604.3,E2 -2604.3} C_VEL
LIN {X 0,Y 565.911,Z 764.636,A -85,B 0,C 180,E1 -2605.728,E2 -2605.728} C_VEL
LIN {X 0,Y 565.866,Z 767.089,A -85,B 0,C 180,E1 -2607.153,E2 -2607.153} C_VEL
LIN {X 0,Y 565.842,Z 768.479,A -85,B 0,C 180,E1 -2608.577,E2 -2608.577} C_VEL
LIN {X 0,Y 565.834,Z 769,A -85,B 0,C 180,E1 -2610.001,E2 -2610.001} C_VEL
LIN {X 0,Y 565.843,Z 768.478,A -85,B 0,C 180,E1 -2611.424,E2 -2611.424} C_VEL
LIN {X 0,Y 565.866,Z 767.086,A -85,B 0,C 180,E1 -2612.848,E2 -2612.848} C_VEL
LIN {X 0,Y 565.911,Z 764.633,A -85,B 0,C 180,E1 -2614.274,E2 -2614.274} C_VEL
LIN {X 0,Y 565.913,Z 760.184,A -85,B 0,C 180,E1 -2616.06,E2 -2616.06} C_VEL
LIN {X 0,Y 565.97,Z 755.466,A -85,B 0,C 180,E1 -2617.493,E2 -2617.493} C_VEL
LIN {X 0,Y 566.011,Z 749.484,A -85,B 0,C 180,E1 -2618.93,E2 -2618.93} C_VEL
LIN {X 0,Y 566.115,Z 741.27,A -85,B 0,C 180,E1 -2620.552,E2 -2620.552} C_VEL
LIN {X 0,Y 566.246,Z 732.442,A -85,B 0,C 180,E1 -2622,E2 -2622} C_VEL
LIN {X 0,Y 566.428,Z 721.905,A -85,B 0,C 180,E1 -2623.453,E2 -2623.453} C_VEL
LIN {X 0,Y 566.662,Z 710.606,A -85,B 0,C 180,E1 -2624.774,E2 -2624.774} C_VEL
LIN {X 0,Y 566.958,Z 698.117,A -85,B 0,C 180,E1 -2626.011,E2 -2626.011} C_VEL
LIN {X 0,Y 567.23,Z 685.046,A -85,B 0,C 180,E1 -2627.114,E2 -2627.114} C_VEL
LIN {X 0,Y 567.567,Z 670.838,A -85,B 0,C 180,E1 -2628.127,E2 -2628.127} C_VEL
LIN {X 0,Y 567.906,Z 655.257,A -85,B 0,C 180,E1 -2629.051,E2 -2629.051} C_VEL
LIN {X 0,Y 568.238,Z 639.895,A -85,B 0,C 180,E1 -2629.795,E2 -2629.795} C_VEL
LIN {X 0,Y 568.53,Z 624.33,A -85,B 0,C 180,E1 -2630.393,E2 -2630.393} C_VEL
LIN {X 0,Y 568.766,Z 608.33,A -85,B 0,C 180,E1 -2630.857,E2 -2630.857} C_VEL
LIN {X 0,Y 568.885,Z 592.509,A -85,B 0,C 180,E1 -2631.182,E2 -2631.182} C_VEL
LIN {X 0,Y 568.778,Z 585.647,A -85,B 0,C 180,E1 -2631.292,E2 -2631.292} C_VEL
LIN {X 0,Y 566.578,Z 577.124,A -85,B 0,C 180,E1 -2631.497,E2 -2631.497} C_VEL
LIN {X 0,Y 566.748,Z 562.746,A -85,B 0,C 180,E1 -2634.546,E2 -2634.546} C_VEL
LIN {X 0,Y 566.975,Z 550.032,A -85,B 0,C 180,E1 -2637.3,E2 -2637.3} C_VEL
LIN {X 0,Y 567.183,Z 537.265,A -85,B 0,C 180,E1 -2640.134,E2 -2640.134} C_VEL
LIN {X 0,Y 567.413,Z 524.604,A -85,B 0,C 180,E1 -2643.024,E2 -2643.024} C_VEL
LIN {X 0,Y 567.632,Z 513.707,A -85,B 0,C 180,E1 -2645.586,E2 -2645.586} C_VEL
LIN {X 0,Y 567.903,Z 501.706,A -85,B 0,C 180,E1 -2648.501,E2 -2648.501} C_VEL
LIN {X 0,Y 567.832,Z 495.54,A -85,B 0,C 180,E1 -2650.061,E2 -2650.061} C_VEL
LIN {X 0,Y 566.215,Z 488.268,A -85,B 0,C 180,E1 -2651.64,E2 -2651.64} C_VEL
LIN {X 0,Y 566.202,Z 488.267,A -85,B 0,C 180,E1 -2654.036,E2 -2654.036} C_VEL
LIN {X 0,Y 566.206,Z 488.269,A -85,B 0,C 180,E1 -2657.083,E2 -2657.083} C_VEL
LIN {X 0,Y 566.228,Z 488.263,A -85,B 0,C 180,E1 -2659.803,E2 -2659.803} C_VEL
LIN {X 0,Y 566.199,Z 488.273,A -85,B 0,C 180,E1 -2662.6,E2 -2662.6} C_VEL
LIN {X 0,Y 566.216,Z 488.264,A -85,B 0,C 180,E1 -2665.183,E2 -2665.183} C_VEL
LIN {X 0,Y 566.231,Z 488.264,A -85,B 0,C 180,E1 -2667.744,E2 -2667.744} C_VEL
LIN {X 0,Y 566.205,Z 488.272,A -85,B 0,C 180,E1 -2670.328,E2 -2670.328} C_VEL
LIN {X 0,Y 566.22,Z 488.265,A -85,B 0,C 180,E1 -2672.662,E2 -2672.662} C_VEL
LIN {X 0,Y 566.238,Z 488.261,A -85,B 0,C 180,E1 -2675.039,E2 -2675.039} C_VEL
LIN {X 0,Y 566.196,Z 488.272,A -85,B 0,C 180,E1 -2678.138,E2 -2678.138} C_VEL
LIN {X 0,Y 566.225,Z 488.265,A -85,B 0,C 180,E1 -2678.685,E2 -2678.685} C_VEL
LIN {X 0,Y 568.119,Z 493.323,A -85,B 0,C 180,E1 -2678.844,E2 -2678.844} C_VEL
LIN {X 0,Y 568.911,Z 495.526,A -85,B 0,C 180,E1 -2678.913,E2 -2678.913} C_VEL
LIN {X 0,Y 568.677,Z 512.14,A -85,B 0,C 180,E1 -2679.283,E2 -2679.283} C_VEL
LIN {X 0,Y 568.439,Z 528.637,A -85,B 0,C 180,E1 -2679.803,E2 -2679.803} C_VEL
LIN {X 0,Y 568.116,Z 545.17,A -85,B 0,C 180,E1 -2680.488,E2 -2680.488} C_VEL
LIN {X 0,Y 567.845,Z 559.567,A -85,B 0,C 180,E1 -2681.229,E2 -2681.229} C_VEL
LIN {X 0,Y 567.527,Z 574.293,A -85,B 0,C 180,E1 -2682.145,E2 -2682.145} C_VEL
LIN {X 0,Y 567.2,Z 588.001,A -85,B 0,C 180,E1 -2683.164,E2 -2683.164} C_VEL
LIN {X 0,Y 566.864,Z 601.558,A -85,B 0,C 180,E1 -2684.356,E2 -2684.356} C_VEL
LIN {X 0,Y 566.623,Z 613.883,A -85,B 0,C 180,E1 -2685.637,E2 -2685.637} C_VEL
LIN {X 0,Y 566.377,Z 624.381,A -85,B 0,C 180,E1 -2686.912,E2 -2686.912} C_VEL
LIN {X 0,Y 566.232,Z 634.536,A -85,B 0,C 180,E1 -2688.364,E2 -2688.364} C_VEL
LIN {X 0,Y 566.122,Z 642.051,A -85,B 0,C 180,E1 -2689.63,E2 -2689.63} C_VEL
LIN {X 0,Y 566.013,Z 649.301,A -85,B 0,C 180,E1 -2691.071,E2 -2691.071} C_VEL
LIN {X 0,Y 565.971,Z 655.3,A -85,B 0,C 180,E1 -2692.508,E2 -2692.508} C_VEL
LIN {X 0,Y 565.915,Z 660.07,A -85,B 0,C 180,E1 -2693.941,E2 -2693.941} C_VEL
LIN {X 0,Y 565.911,Z 664.549,A -85,B 0,C 180,E1 -2695.727,E2 -2695.727} C_VEL
LIN {X 0,Y 565.872,Z 667.025,A -85,B 0,C 180,E1 -2697.153,E2 -2697.153} C_VEL
LIN {X 0,Y 565.839,Z 668.462,A -85,B 0,C 180,E1 -2698.577,E2 -2698.577} C_VEL
LIN {X 0,Y 565.836,Z 668.996,A -85,B 0,C 180,E1 -2700,E2 -2700} C_VEL
LIN {X 0,Y 565.839,Z 668.52,A -85,B 0,C 180,E1 -2701.424,E2 -2701.424} C_VEL
LIN {X 0,Y 565.872,Z 667.138,A -85,B 0,C 180,E1 -2702.848,E2 -2702.848} C_VEL
LIN {X 0,Y 565.911,Z 664.733,A -85,B 0,C 180,E1 -2704.274,E2 -2704.274} C_VEL
LIN {X 0,Y 565.917,Z 660.332,A -85,B 0,C 180,E1 -2706.06,E2 -2706.06} C_VEL
LIN {X 0,Y 565.972,Z 655.62,A -85,B 0,C 180,E1 -2707.492,E2 -2707.492} C_VEL
LIN {X 0,Y 566.006,Z 649.692,A -85,B 0,C 180,E1 -2708.929,E2 -2708.929} C_VEL
LIN {X 0,Y 566.115,Z 641.542,A -85,B 0,C 180,E1 -2710.551,E2 -2710.551} C_VEL
LIN {X 0,Y 566.248,Z 632.764,A -85,B 0,C 180,E1 -2711.999,E2 -2711.999} C_VEL
LIN {X 0,Y 566.421,Z 622.268,A -85,B 0,C 180,E1 -2713.453,E2 -2713.453} C_VEL
LIN {X 0,Y 566.67,Z 610.713,A -85,B 0,C 180,E1 -2714.806,E2 -2714.806} C_VEL
LIN {X 0,Y 566.935,Z 598.605,A -85,B 0,C 180,E1 -2716.011,E2 -2716.011} C_VEL
LIN {X 0,Y 567.213,Z 585.619,A -85,B 0,C 180,E1 -2717.114,E2 -2717.114} C_VEL
LIN {X 0,Y 567.568,Z 571.552,A -85,B 0,C 180,E1 -2718.127,E2 -2718.127} C_VEL
LIN {X 0,Y 567.886,Z 556.117,A -85,B 0,C 180,E1 -2719.051,E2 -2719.051} C_VEL
LIN {X 0,Y 568.25,Z 540.188,A -85,B 0,C 180,E1 -2719.827,E2 -2719.827} C_VEL
LIN {X 0,Y 568.543,Z 522.895,A -85,B 0,C 180,E1 -2720.487,E2 -2720.487} C_VEL
LIN {X 0,Y 568.59,Z 520.064,A -85,B 0,C 180,E1 -2720.573,E2 -2720.573} C_VEL
LIN {X 0,Y 568.441,Z 514.374,A -85,B 0,C 180,E1 -2720.754,E2 -2720.754} C_VEL
LIN {X 0,Y 567.378,Z 508.806,A -85,B 0,C 180,E1 -2720.945,E2 -2720.945} C_VEL
LIN {X 0,Y 566.267,Z 505.192,A -85,B 0,C 180,E1 -2721.074,E2 -2721.074} C_VEL
LIN {X 0,Y 563.406,Z 498.14,A -85,B 0,C 180,E1 -2721.344,E2 -2721.344} C_VEL
LIN {X 0,Y 559.84,Z 491.363,A -85,B 0,C 180,E1 -2721.604,E2 -2721.604} C_VEL
LIN {X 0,Y 559.164,Z 489.148,A -85,B 0,C 180,E1 -2721.678,E2 -2721.678} C_VEL
LIN {X 0,Y 559.161,Z 489.15,A -85,B 0,C 180,E1 -2724.505,E2 -2724.505} C_VEL
LIN {X 0,Y 559.172,Z 489.145,A -85,B 0,C 180,E1 -2726.903,E2 -2726.903} C_VEL
LIN {X 0,Y 559.153,Z 489.147,A -85,B 0,C 180,E1 -2729.858,E2 -2729.858} C_VEL
LIN {X 0,Y 559.161,Z 489.146,A -85,B 0,C 180,E1 -2732.715,E2 -2732.715} C_VEL
LIN {X 0,Y 559.153,Z 489.146,A -85,B 0,C 180,E1 -2735.323,E2 -2735.323} C_VEL
LIN {X 0,Y 559.138,Z 489.148,A -85,B 0,C 180,E1 -2738.018,E2 -2738.018} C_VEL
LIN {X 0,Y 559.159,Z 489.146,A -85,B 0,C 180,E1 -2740.813,E2 -2740.813} C_VEL
LIN {X 0,Y 559.143,Z 489.148,A -85,B 0,C 180,E1 -2743.734,E2 -2743.734} C_VEL
LIN {X 0,Y 559.155,Z 489.146,A -85,B 0,C 180,E1 -2746.803,E2 -2746.803} C_VEL
LIN {X 0,Y 559.181,Z 489.145,A -85,B 0,C 180,E1 -2749.189,E2 -2749.189} C_VEL
LIN {X 0,Y 559.139,Z 489.151,A -85,B 0,C 180,E1 -2751.982,E2 -2751.982} C_VEL
LIN {X 0,Y 559.137,Z 489.152,A -85,B 0,C 180,E1 -2754.787,E2 -2754.787} C_VEL
LIN {X 0,Y 559.162,Z 489.15,A -85,B 0,C 180,E1 -2757.364,E2 -2757.364} C_VEL
LIN {X 0,Y 559.154,Z 489.15,A -85,B 0,C 180,E1 -2760.143,E2 -2760.143} C_VEL
LIN {X 0,Y 559.176,Z 489.148,A -85,B 0,C 180,E1 -2763.097,E2 -2763.097} C_VEL
LIN {X 0,Y 559.187,Z 489.251,A -85,B 0,C 180,E1 -2765.989,E2 -2765.989} C_VEL
LIN {X 0,Y 559.17,Z 494.276,A -85,B 0,C 180,E1 -2768.623,E2 -2768.623} C_VEL
LIN {X 0,Y 559.139,Z 498.539,A -85,B 0,C 180,E1 -2770.925,E2 -2770.925} C_VEL
LIN {X 0,Y 559.099,Z 502.632,A -85,B 0,C 180,E1 -2773.194,E2 -2773.194} C_VEL
LIN {X 0,Y 559.08,Z 506.694,A -85,B 0,C 180,E1 -2775.454,E2 -2775.454} C_VEL
LIN {X 0,Y 559.047,Z 512.741,A -85,B 0,C 180,E1 -2778.689,E2 -2778.689} C_VEL
LIN {X 0,Y 558.965,Z 519.21,A -85,B 0,C 180,E1 -2782.05,E2 -2782.05} C_VEL
LIN {X 0,Y 558.943,Z 521.662,A -85,B 0,C 180,E1 -2783.302,E2 -2783.302} C_VEL
LIN {X 0,Y 562.266,Z 533.633,A -85,B 0,C 180,E1 -2783.622,E2 -2783.622} C_VEL
LIN {X 0,Y 562.085,Z 550.078,A -85,B 0,C 180,E1 -2783.972,E2 -2783.972} C_VEL
LIN {X 0,Y 561.77,Z 567.881,A -85,B 0,C 180,E1 -2784.525,E2 -2784.525} C_VEL
LIN {X 0,Y 561.43,Z 583.15,A -85,B 0,C 180,E1 -2785.152,E2 -2785.152} C_VEL
LIN {X 0,Y 561.131,Z 597.296,A -85,B 0,C 180,E1 -2785.869,E2 -2785.869} C_VEL
LIN {X 0,Y 560.743,Z 612.012,A -85,B 0,C 180,E1 -2786.766,E2 -2786.766} C_VEL
LIN {X 0,Y 560.367,Z 626.62,A -85,B 0,C 180,E1 -2787.843,E2 -2787.843} C_VEL
LIN {X 0,Y 560.022,Z 639.042,A -85,B 0,C 180,E1 -2788.921,E2 -2788.921} C_VEL
LIN {X 0,Y 559.699,Z 651.474,A -85,B 0,C 180,E1 -2790.179,E2 -2790.179} C_VEL
LIN {X 0,Y 559.386,Z 663.407,A -85,B 0,C 180,E1 -2791.619,E2 -2791.619} C_VEL
LIN {X 0,Y 559.213,Z 672.353,A -85,B 0,C 180,E1 -2792.881,E2 -2792.881} C_VEL
LIN {X 0,Y 559.076,Z 681.086,A -85,B 0,C 180,E1 -2794.325,E2 -2794.325} C_VEL
LIN {X 0,Y 558.953,Z 688.482,A -85,B 0,C 180,E1 -2795.772,E2 -2795.772} C_VEL
LIN {X 0,Y 558.893,Z 694.574,A -85,B 0,C 180,E1 -2797.223,E2 -2797.223} C_VEL
LIN {X 0,Y 558.825,Z 699.516,A -85,B 0,C 180,E1 -2798.679,E2 -2798.679} C_VEL
LIN {X 0,Y 558.794,Z 703.415,A -85,B 0,C 180,E1 -2800.141,E2 -2800.141} C_VEL
LIN {X 0,Y 558.773,Z 706.226,A -85,B 0,C 180,E1 -2801.609,E2 -2801.609} C_VEL
LIN {X 0,Y 558.739,Z 708.081,A -85,B 0,C 180,E1 -2803.085,E2 -2803.085} C_VEL
LIN {X 0,Y 558.727,Z 708.903,A -85,B 0,C 180,E1 -2804.57,E2 -2804.57} C_VEL
LIN {X 0,Y 558.722,Z 708.745,A -85,B 0,C 180,E1 -2806.064,E2 -2806.064} C_VEL
LIN {X 0,Y 558.745,Z 707.507,A -85,B 0,C 180,E1 -2807.569,E2 -2807.569} C_VEL
LIN {X 0,Y 558.774,Z 704.626,A -85,B 0,C 180,E1 -2809.383,E2 -2809.383} C_VEL
LIN {X 0,Y 558.833,Z 700.701,A -85,B 0,C 180,E1 -2811.002,E2 -2811.002} C_VEL
LIN {X 0,Y 558.881,Z 695.725,A -85,B 0,C 180,E1 -2812.552,E2 -2812.552} C_VEL
LIN {X 0,Y 558.951,Z 689.368,A -85,B 0,C 180,E1 -2814.118,E2 -2814.118} C_VEL
LIN {X 0,Y 559.038,Z 681.436,A -85,B 0,C 180,E1 -2815.703,E2 -2815.703} C_VEL
LIN {X 0,Y 559.201,Z 673.056,A -85,B 0,C 180,E1 -2817.102,E2 -2817.102} C_VEL
LIN {X 0,Y 559.4,Z 663.077,A -85,B 0,C 180,E1 -2818.515,E2 -2818.515} C_VEL
LIN {X 0,Y 559.75,Z 650.979,A -85,B 0,C 180,E1 -2819.964,E2 -2819.964} C_VEL
LIN {X 0,Y 559.994,Z 639.645,A -85,B 0,C 180,E1 -2821.114,E2 -2821.114} C_VEL
LIN {X 0,Y 560.333,Z 627.07,A -85,B 0,C 180,E1 -2822.211,E2 -2822.211} C_VEL
LIN {X 0,Y 560.718,Z 612.569,A -85,B 0,C 180,E1 -2823.287,E2 -2823.287} C_VEL
LIN {X 0,Y 561.086,Z 596.998,A -85,B 0,C 180,E1 -2824.238,E2 -2824.238} C_VEL
LIN {X 0,Y 561.409,Z 583.146,A -85,B 0,C 180,E1 -2824.939,E2 -2824.939} C_VEL
LIN {X 0,Y 561.725,Z 568.6,A -85,B 0,C 180,E1 -2825.539,E2 -2825.539} C_VEL
LIN {X 0,Y 562.04,Z 551.188,A -85,B 0,C 180,E1 -2826.09,E2 -2826.09} C_VEL
LIN {X 0,Y 562.268,Z 535.01,A -85,B 0,C 180,E1 -2826.444,E2 -2826.444} C_VEL
LIN {X 0,Y 561.954,Z 532.212,A -85,B 0,C 180,E1 -2826.504,E2 -2826.504} C_VEL
LIN {X 0,Y 558.939,Z 521.638,A -85,B 0,C 180,E1 -2826.8,E2 -2826.8} C_VEL
LIN {X 0,Y 558.93,Z 515.592,A -85,B 0,C 180,E1 -2829.913,E2 -2829.913} C_VEL
LIN {X 0,Y 559.005,Z 510.191,A -85,B 0,C 180,E1 -2832.756,E2 -2832.756} C_VEL
LIN {X 0,Y 559.067,Z 504.623,A -85,B 0,C 180,E1 -2835.768,E2 -2835.768} C_VEL
LIN {X 0,Y 559.13,Z 498.904,A -85,B 0,C 180,E1 -2838.951,E2 -2838.951} C_VEL
LIN {X 0,Y 559.114,Z 493.219,A -85,B 0,C 180,E1 -2841.98,E2 -2841.98} C_VEL
LIN {X 0,Y 559.178,Z 489.149,A -85,B 0,C 180,E1 -2844.126,E2 -2844.126} C_VEL
LIN {X 0,Y 559.172,Z 489.148,A -85,B 0,C 180,E1 -2846.425,E2 -2846.425} C_VEL
LIN {X 0,Y 559.159,Z 489.148,A -85,B 0,C 180,E1 -2848.981,E2 -2848.981} C_VEL
LIN {X 0,Y 559.163,Z 489.146,A -85,B 0,C 180,E1 -2851.617,E2 -2851.617} C_VEL
LIN {X 0,Y 559.193,Z 489.143,A -85,B 0,C 180,E1 -2853.903,E2 -2853.903} C_VEL
LIN {X 0,Y 559.155,Z 489.147,A -85,B 0,C 180,E1 -2857.068,E2 -2857.068} C_VEL
LIN {X 0,Y 559.177,Z 489.145,A -85,B 0,C 180,E1 -2859.395,E2 -2859.395} C_VEL
LIN {X 0,Y 559.149,Z 489.151,A -85,B 0,C 180,E1 -2861.685,E2 -2861.685} C_VEL
LIN {X 0,Y 559.162,Z 489.145,A -85,B 0,C 180,E1 -2863.947,E2 -2863.947} C_VEL
LIN {X 0,Y 559.167,Z 489.145,A -85,B 0,C 180,E1 -2866.184,E2 -2866.184} C_VEL
LIN {X 0,Y 559.202,Z 489.139,A -85,B 0,C 180,E1 -2869.133,E2 -2869.133} C_VEL
LIN {X 0,Y 559.201,Z 489.14,A -85,B 0,C 180,E1 -2872.053,E2 -2872.053} C_VEL
LIN {X 0,Y 559.256,Z 489.135,A -85,B 0,C 180,E1 -2874.953,E2 -2874.953} C_VEL
LIN {X 0,Y 559.25,Z 489.138,A -85,B 0,C 180,E1 -2877.839,E2 -2877.839} C_VEL
LIN {X 0,Y 559.27,Z 489.136,A -85,B 0,C 180,E1 -2880.72,E2 -2880.72} C_VEL
LIN {X 0,Y 559.236,Z 489.136,A -85,B 0,C 180,E1 -2882.881,E2 -2882.881} C_VEL
LIN {X 0,Y 559.221,Z 489.137,A -85,B 0,C 180,E1 -2885.77,E2 -2885.77} C_VEL
LIN {X 0,Y 559.194,Z 489.143,A -85,B 0,C 180,E1 -2888.674,E2 -2888.674} C_VEL
LIN {X 0,Y 559.198,Z 489.143,A -85,B 0,C 180,E1 -2891.6,E2 -2891.6} C_VEL
LIN {X 0,Y 559.187,Z 489.143,A -85,B 0,C 180,E1 -2894.596,E2 -2894.596} C_VEL
LIN {X 0,Y 559.153,Z 489.138,A -85,B 0,C 180,E1 -2897.557,E2 -2897.557} C_VEL
LIN {X 0,Y 559.164,Z 489.148,A -85,B 0,C 180,E1 -2899.837,E2 -2899.837} C_VEL
LIN {X 0,Y 559.145,Z 489.15,A -85,B 0,C 180,E1 -2902.152,E2 -2902.152} C_VEL
LIN {X 0,Y 559.15,Z 489.139,A -85,B 0,C 180,E1 -2904.505,E2 -2904.505} C_VEL
LIN {X 0,Y 559.17,Z 489.145,A -85,B 0,C 180,E1 -2906.902,E2 -2906.902} C_VEL
LIN {X 0,Y 559.179,Z 489.144,A -85,B 0,C 180,E1 -2909.866,E2 -2909.866} C_VEL
LIN {X 0,Y 559.166,Z 489.145,A -85,B 0,C 180,E1 -2912.714,E2 -2912.714} C_VEL
LIN {X 0,Y 559.15,Z 489.147,A -85,B 0,C 180,E1 -2915.322,E2 -2915.322} C_VEL
LIN {X 0,Y 559.126,Z 489.15,A -85,B 0,C 180,E1 -2918.018,E2 -2918.018} C_VEL
LIN {X 0,Y 559.171,Z 489.144,A -85,B 0,C 180,E1 -2920.811,E2 -2920.811} C_VEL
LIN {X 0,Y 559.153,Z 489.148,A -85,B 0,C 180,E1 -2923.732,E2 -2923.732} C_VEL
LIN {X 0,Y 559.165,Z 489.149,A -85,B 0,C 180,E1 -2926.801,E2 -2926.801} C_VEL
LIN {X 0,Y 559.194,Z 489.186,A -85,B 0,C 180,E1 -2927.756,E2 -2927.756} C_VEL
LIN {X 0,Y 560.971,Z 497.169,A -85,B 0,C 180,E1 -2929.838,E2 -2929.838} C_VEL
LIN {X 0,Y 561.114,Z 502.817,A -85,B 0,C 180,E1 -2931.227,E2 -2931.227} C_VEL
LIN {X 0,Y 560.858,Z 513.714,A -85,B 0,C 180,E1 -2933.919,E2 -2933.919} C_VEL
LIN {X 0,Y 560.534,Z 526.161,A -85,B 0,C 180,E1 -2936.886,E2 -2936.886} C_VEL
LIN {X 0,Y 560.261,Z 539.142,A -85,B 0,C 180,E1 -2939.884,E2 -2939.884} C_VEL
LIN {X 0,Y 560.047,Z 551.767,A -85,B 0,C 180,E1 -2942.721,E2 -2942.721} C_VEL
LIN {X 0,Y 559.769,Z 564.57,A -85,B 0,C 180,E1 -2945.525,E2 -2945.525} C_VEL
LIN {X 0,Y 559.611,Z 577.095,A -85,B 0,C 180,E1 -2948.216,E2 -2948.216} C_VEL
LIN {X 0,Y 562.261,Z 587.374,A -85,B 0,C 180,E1 -2948.474,E2 -2948.474} C_VEL
LIN {X 0,Y 562.144,Z 604.665,A -85,B 0,C 180,E1 -2948.792,E2 -2948.792} C_VEL
LIN {X 0,Y 561.93,Z 620.762,A -85,B 0,C 180,E1 -2949.239,E2 -2949.239} C_VEL
LIN {X 0,Y 561.579,Z 636.539,A -85,B 0,C 180,E1 -2949.818,E2 -2949.818} C_VEL
LIN {X 0,Y 561.238,Z 651.782,A -85,B 0,C 180,E1 -2950.525,E2 -2950.525} C_VEL
LIN {X 0,Y 560.882,Z 666.588,A -85,B 0,C 180,E1 -2951.367,E2 -2951.367} C_VEL
LIN {X 0,Y 560.467,Z 681.087,A -85,B 0,C 180,E1 -2952.364,E2 -2952.364} C_VEL
LIN {X 0,Y 560.157,Z 693.988,A -85,B 0,C 180,E1 -2953.416,E2 -2953.416} C_VEL
LIN {X 0,Y 559.856,Z 705.737,A -85,B 0,C 180,E1 -2954.53,E2 -2954.53} C_VEL
LIN {X 0,Y 559.588,Z 717.452,A -85,B 0,C 180,E1 -2955.825,E2 -2955.825} C_VEL
LIN {X 0,Y 559.3,Z 728.739,A -85,B 0,C 180,E1 -2957.298,E2 -2957.298} C_VEL
LIN {X 0,Y 559.159,Z 738.238,A -85,B 0,C 180,E1 -2958.777,E2 -2958.777} C_VEL
LIN {X 0,Y 558.973,Z 746.054,A -85,B 0,C 180,E1 -2960.228,E2 -2960.228} C_VEL
LIN {X 0,Y 558.916,Z 752.628,A -85,B 0,C 180,E1 -2961.686,E2 -2961.686} C_VEL
LIN {X 0,Y 558.878,Z 757.961,A -85,B 0,C 180,E1 -2963.14,E2 -2963.14} C_VEL
LIN {X 0,Y 558.861,Z 761.249,A -85,B 0,C 180,E1 -2964.227,E2 -2964.227} C_VEL
LIN {X 0,Y 558.805,Z 764.637,A -85,B 0,C 180,E1 -2965.673,E2 -2965.673} C_VEL
LIN {X 0,Y 558.787,Z 767.089,A -85,B 0,C 180,E1 -2967.117,E2 -2967.117} C_VEL
LIN {X 0,Y 558.742,Z 768.479,A -85,B 0,C 180,E1 -2968.559,E2 -2968.559} C_VEL
LIN {X 0,Y 558.735,Z 769,A -85,B 0,C 180,E1 -2970.001,E2 -2970.001} C_VEL
LIN {X 0,Y 558.742,Z 768.478,A -85,B 0,C 180,E1 -2971.442,E2 -2971.442} C_VEL
LIN {X 0,Y 558.788,Z 767.086,A -85,B 0,C 180,E1 -2972.884,E2 -2972.884} C_VEL
LIN {X 0,Y 558.806,Z 764.633,A -85,B 0,C 180,E1 -2974.328,E2 -2974.328} C_VEL
LIN {X 0,Y 558.862,Z 761.246,A -85,B 0,C 180,E1 -2975.775,E2 -2975.775} C_VEL
LIN {X 0,Y 558.895,Z 755.466,A -85,B 0,C 180,E1 -2977.588,E2 -2977.588} C_VEL
LIN {X 0,Y 558.939,Z 747.854,A -85,B 0,C 180,E1 -2979.408,E2 -2979.408} C_VEL
LIN {X 0,Y 559.116,Z 739.273,A -85,B 0,C 180,E1 -2981.047,E2 -2981.047} C_VEL
LIN {X 0,Y 559.276,Z 729.967,A -85,B 0,C 180,E1 -2982.52,E2 -2982.52} C_VEL
LIN {X 0,Y 559.471,Z 720.419,A -85,B 0,C 180,E1 -2983.809,E2 -2983.809} C_VEL
LIN {X 0,Y 559.793,Z 709.253,A -85,B 0,C 180,E1 -2985.103,E2 -2985.103} C_VEL
LIN {X 0,Y 560.051,Z 697.136,A -85,B 0,C 180,E1 -2986.307,E2 -2986.307} C_VEL
LIN {X 0,Y 560.408,Z 683.872,A -85,B 0,C 180,E1 -2987.423,E2 -2987.423} C_VEL
LIN {X 0,Y 560.801,Z 669.425,A -85,B 0,C 180,E1 -2988.448,E2 -2988.448} C_VEL
LIN {X 0,Y 561.155,Z 655.258,A -85,B 0,C 180,E1 -2989.289,E2 -2989.289} C_VEL
LIN {X 0,Y 561.537,Z 639.896,A -85,B 0,C 180,E1 -2990.041,E2 -2990.041} C_VEL
LIN {X 0,Y 561.868,Z 624.33,A -85,B 0,C 180,E1 -2990.646,E2 -2990.646} C_VEL
LIN {X 0,Y 562.14,Z 608.33,A -85,B 0,C 180,E1 -2991.114,E2 -2991.114} C_VEL
LIN {X 0,Y 562.267,Z 592.375,A -85,B 0,C 180,E1 -2991.446,E2 -2991.446} C_VEL
LIN {X 0,Y 562.148,Z 586.793,A -85,B 0,C 180,E1 -2991.54,E2 -2991.54} C_VEL
LIN {X 0,Y 559.598,Z 577.076,A -85,B 0,C 180,E1 -2991.789,E2 -2991.789} C_VEL
LIN {X 0,Y 559.764,Z 564.562,A -85,B 0,C 180,E1 -2994.477,E2 -2994.477} C_VEL
LIN {X 0,Y 560.042,Z 551.765,A -85,B 0,C 180,E1 -2997.28,E2 -2997.28} C_VEL
LIN {X 0,Y 560.266,Z 539.135,A -85,B 0,C 180,E1 -3000.117,E2 -3000.117} C_VEL
LIN {X 0,Y 560.54,Z 526.154,A -85,B 0,C 180,E1 -3003.115,E2 -3003.115} C_VEL
LIN {X 0,Y 560.818,Z 515.246,A -85,B 0,C 180,E1 -3005.71,E2 -3005.71} C_VEL
LIN {X 0,Y 561.112,Z 504.627,A -85,B 0,C 180,E1 -3008.316,E2 -3008.316} C_VEL
LIN {X 0,Y 561.108,Z 498.931,A -85,B 0,C 180,E1 -3009.702,E2 -3009.702} C_VEL
LIN {X 0,Y 559.794,Z 492.127,A -85,B 0,C 180,E1 -3011.125,E2 -3011.125} C_VEL
LIN {X 0,Y 559.193,Z 489.143,A -85,B 0,C 180,E1 -3011.768,E2 -3011.768} C_VEL
LIN {X 0,Y 559.142,Z 489.152,A -85,B 0,C 180,E1 -3014.739,E2 -3014.739} C_VEL
LIN {X 0,Y 559.161,Z 489.145,A -85,B 0,C 180,E1 -3017.257,E2 -3017.257} C_VEL
LIN {X 0,Y 559.187,Z 489.143,A -85,B 0,C 180,E1 -3020.135,E2 -3020.135} C_VEL
LIN {X 0,Y 559.144,Z 489.148,A -85,B 0,C 180,E1 -3022.892,E2 -3022.892} C_VEL
LIN {X 0,Y 559.154,Z 489.144,A -85,B 0,C 180,E1 -3025.556,E2 -3025.556} C_VEL
LIN {X 0,Y 559.166,Z 489.149,A -85,B 0,C 180,E1 -3028.138,E2 -3028.138} C_VEL
LIN {X 0,Y 559.145,Z 489.147,A -85,B 0,C 180,E1 -3030.647,E2 -3030.647} C_VEL
LIN {X 0,Y 559.173,Z 489.141,A -85,B 0,C 180,E1 -3033.173,E2 -3033.173} C_VEL
LIN {X 0,Y 559.159,Z 489.146,A -85,B 0,C 180,E1 -3035.495,E2 -3035.495} C_VEL
LIN {X 0,Y 559.169,Z 489.145,A -85,B 0,C 180,E1 -3038.418,E2 -3038.418} C_VEL
LIN {X 0,Y 560.963,Z 493.963,A -85,B 0,C 180,E1 -3038.57,E2 -3038.57} C_VEL
LIN {X 0,Y 562.22,Z 496.915,A -85,B 0,C 180,E1 -3038.676,E2 -3038.676} C_VEL
LIN {X 0,Y 562.027,Z 513.945,A -85,B 0,C 180,E1 -3039.074,E2 -3039.074} C_VEL
LIN {X 0,Y 561.754,Z 530.436,A -85,B 0,C 180,E1 -3039.619,E2 -3039.619} C_VEL
LIN {X 0,Y 561.395,Z 545.188,A -85,B 0,C 180,E1 -3040.245,E2 -3040.245} C_VEL
LIN {X 0,Y 561.076,Z 559.573,A -85,B 0,C 180,E1 -3040.994,E2 -3040.994} C_VEL
LIN {X 0,Y 560.692,Z 574.682,A -85,B 0,C 180,E1 -3041.946,E2 -3041.946} C_VEL
LIN {X 0,Y 560.299,Z 588.013,A -85,B 0,C 180,E1 -3042.951,E2 -3042.951} C_VEL
LIN {X 0,Y 559.937,Z 601.566,A -85,B 0,C 180,E1 -3044.158,E2 -3044.158} C_VEL
LIN {X 0,Y 559.661,Z 613.891,A -85,B 0,C 180,E1 -3045.455,E2 -3045.455} C_VEL
LIN {X 0,Y 559.386,Z 624.389,A -85,B 0,C 180,E1 -3046.745,E2 -3046.745} C_VEL
LIN {X 0,Y 559.211,Z 634.541,A -85,B 0,C 180,E1 -3048.216,E2 -3048.216} C_VEL
LIN {X 0,Y 559.078,Z 642.058,A -85,B 0,C 180,E1 -3049.498,E2 -3049.498} C_VEL
LIN {X 0,Y 558.949,Z 649.306,A -85,B 0,C 180,E1 -3050.958,E2 -3050.958} C_VEL
LIN {X 0,Y 558.896,Z 655.303,A -85,B 0,C 180,E1 -3052.413,E2 -3052.413} C_VEL
LIN {X 0,Y 558.864,Z 661.118,A -85,B 0,C 180,E1 -3054.226,E2 -3054.226} C_VEL
LIN {X 0,Y 558.805,Z 664.551,A -85,B 0,C 180,E1 -3055.673,E2 -3055.673} C_VEL
LIN {X 0,Y 558.793,Z 667.024,A -85,B 0,C 180,E1 -3057.117,E2 -3057.117} C_VEL
LIN {X 0,Y 558.738,Z 668.465,A -85,B 0,C 180,E1 -3058.559,E2 -3058.559} C_VEL
LIN {X 0,Y 558.737,Z 668.996,A -85,B 0,C 180,E1 -3060,E2 -3060} C_VEL
LIN {X 0,Y 558.738,Z 668.522,A -85,B 0,C 180,E1 -3061.442,E2 -3061.442} C_VEL
LIN {X 0,Y 558.793,Z 667.136,A -85,B 0,C 180,E1 -3062.884,E2 -3062.884} C_VEL
LIN {X 0,Y 558.805,Z 664.734,A -85,B 0,C 180,E1 -3064.328,E2 -3064.328} C_VEL
LIN {X 0,Y 558.865,Z 661.365,A -85,B 0,C 180,E1 -3065.774,E2 -3065.774} C_VEL
LIN {X 0,Y 558.892,Z 656.89,A -85,B 0,C 180,E1 -3067.224,E2 -3067.224} C_VEL
LIN {X 0,Y 558.933,Z 651.309,A -85,B 0,C 180,E1 -3068.679,E2 -3068.679} C_VEL
LIN {X 0,Y 559.025,Z 644.469,A -85,B 0,C 180,E1 -3070.138,E2 -3070.138} C_VEL
LIN {X 0,Y 559.187,Z 635.101,A -85,B 0,C 180,E1 -3071.785,E2 -3071.785} C_VEL
LIN {X 0,Y 559.391,Z 625.031,A -85,B 0,C 180,E1 -3073.255,E2 -3073.255} C_VEL
LIN {X 0,Y 559.641,Z 613.95,A -85,B 0,C 180,E1 -3074.63,E2 -3074.63} C_VEL
LIN {X 0,Y 559.919,Z 602.498,A -85,B 0,C 180,E1 -3075.843,E2 -3075.843} C_VEL
LIN {X 0,Y 560.274,Z 589.086,A -85,B 0,C 180,E1 -3077.051,E2 -3077.051} C_VEL
LIN {X 0,Y 560.638,Z 575.667,A -85,B 0,C 180,E1 -3078.075,E2 -3078.075} C_VEL
LIN {X 0,Y 561.022,Z 561.075,A -85,B 0,C 180,E1 -3079.009,E2 -3079.009} C_VEL
LIN {X 0,Y 561.418,Z 545.578,A -85,B 0,C 180,E1 -3079.825,E2 -3079.825} C_VEL
LIN {X 0,Y 561.694,Z 531.089,A -85,B 0,C 180,E1 -3080.444,E2 -3080.444} C_VEL
LIN {X 0,Y 561.968,Z 516.742,A -85,B 0,C 180,E1 -3080.929,E2 -3080.929} C_VEL
LIN {X 0,Y 562.218,Z 500.82,A -85,B 0,C 180,E1 -3081.334,E2 -3081.334} C_VEL
LIN {X 0,Y 562.123,Z 496.725,A -85,B 0,C 180,E1 -3081.421,E2 -3081.421} C_VEL
LIN {X 0,Y 559.84,Z 491.363,A -85,B 0,C 180,E1 -3081.604,E2 -3081.604} C_VEL
LIN {X 0,Y 558.565,Z 489.983,A -85,B 0,C 180,E1 -3081.751,E2 -3081.751} C_VEL
LIN {X 0,Y 556.889,Z 489.482,A -85,B 0,C 180,E1 -3082.05,E2 -3082.05} C_VEL
LIN {X 0,Y 554.548,Z 489.722,A -85,B 0,C 180,E1 -3082.699,E2 -3082.699} C_VEL
LIN {X 0,Y 553.198,Z 490.135,A -85,B 0,C 180,E1 -3083.35,E2 -3083.35} C_VEL
LIN {X 0,Y 552.213,Z 490.093,A -85,B 0,C 180,E1 -3084.28,E2 -3084.28} C_VEL
LIN {X 0,Y 552.111,Z 490.026,A -85,B 0,C 180,E1 -3084.749,E2 -3084.749} C_VEL
LIN {X 0,Y 552.133,Z 490.024,A -85,B 0,C 180,E1 -3087.274,E2 -3087.274} C_VEL
LIN {X 0,Y 552.121,Z 490.025,A -85,B 0,C 180,E1 -3090.051,E2 -3090.051} C_VEL
LIN {X 0,Y 552.119,Z 490.024,A -85,B 0,C 180,E1 -3092.847,E2 -3092.847} C_VEL
LIN {X 0,Y 552.104,Z 490.025,A -85,B 0,C 180,E1 -3095.443,E2 -3095.443} C_VEL
LIN {X 0,Y 552.101,Z 490.026,A -85,B 0,C 180,E1 -3097.886,E2 -3097.886} C_VEL
LIN {X 0,Y 552.114,Z 490.027,A -85,B 0,C 180,E1 -3100.481,E2 -3100.481} C_VEL
LIN {X 0,Y 552.111,Z 490.026,A -85,B 0,C 180,E1 -3103.424,E2 -3103.424} C_VEL
LIN {X 0,Y 552.112,Z 490.024,A -85,B 0,C 180,E1 -3106.576,E2 -3106.576} C_VEL
LIN {X 0,Y 552.126,Z 490.022,A -85,B 0,C 180,E1 -3109.52,E2 -3109.52} C_VEL
LIN {X 0,Y 552.098,Z 490.026,A -85,B 0,C 180,E1 -3112.336,E2 -3112.336} C_VEL
LIN {X 0,Y 552.089,Z 490.028,A -85,B 0,C 180,E1 -3115.051,E2 -3115.051} C_VEL
LIN {X 0,Y 552.122,Z 490.027,A -85,B 0,C 180,E1 -3117.681,E2 -3117.681} C_VEL
LIN {X 0,Y 552.117,Z 490.028,A -85,B 0,C 180,E1 -3120.235,E2 -3120.235} C_VEL
LIN {X 0,Y 552.145,Z 490.023,A -85,B 0,C 180,E1 -3123,E2 -3123} C_VEL
LIN {X 0,Y 552.165,Z 490.133,A -85,B 0,C 180,E1 -3125.964,E2 -3125.964} C_VEL
LIN {X 0,Y 552.085,Z 496.105,A -85,B 0,C 180,E1 -3129.118,E2 -3129.118} C_VEL
LIN {X 0,Y 552.075,Z 500.361,A -85,B 0,C 180,E1 -3131.442,E2 -3131.442} C_VEL
LIN {X 0,Y 552.01,Z 504.451,A -85,B 0,C 180,E1 -3133.733,E2 -3133.733} C_VEL
LIN {X 0,Y 552.009,Z 508.446,A -85,B 0,C 180,E1 -3136.001,E2 -3136.001} C_VEL
LIN {X 0,Y 551.956,Z 513.986,A -85,B 0,C 180,E1 -3138.989,E2 -3138.989} C_VEL
LIN {X 0,Y 551.91,Z 519.611,A -85,B 0,C 180,E1 -3141.947,E2 -3141.947} C_VEL
LIN {X 0,Y 551.885,Z 521.677,A -85,B 0,C 180,E1 -3143.013,E2 -3143.013} C_VEL
LIN {X 0,Y 554.14,Z 529.436,A -85,B 0,C 180,E1 -3143.221,E2 -3143.221} C_VEL
LIN {X 0,Y 555.629,Z 534.64,A -85,B 0,C 180,E1 -3143.371,E2 -3143.371} C_VEL
LIN {X 0,Y 555.45,Z 551.459,A -85,B 0,C 180,E1 -3143.745,E2 -3143.745} C_VEL
LIN {X 0,Y 555.085,Z 568.142,A -85,B 0,C 180,E1 -3144.277,E2 -3144.277} C_VEL
LIN {X 0,Y 554.708,Z 583.356,A -85,B 0,C 180,E1 -3144.911,E2 -3144.911} C_VEL
LIN {X 0,Y 554.36,Z 597.485,A -85,B 0,C 180,E1 -3145.637,E2 -3145.637} C_VEL
LIN {X 0,Y 553.924,Z 612.183,A -85,B 0,C 180,E1 -3146.544,E2 -3146.544} C_VEL
LIN {X 0,Y 553.487,Z 626.754,A -85,B 0,C 180,E1 -3147.634,E2 -3147.634} C_VEL
LIN {X 0,Y 553.115,Z 639.155,A -85,B 0,C 180,E1 -3148.725,E2 -3148.725} C_VEL
LIN {X 0,Y 552.754,Z 651.574,A -85,B 0,C 180,E1 -3149.999,E2 -3149.999} C_VEL
LIN {X 0,Y 552.39,Z 663.487,A -85,B 0,C 180,E1 -3151.457,E2 -3151.457} C_VEL
LIN {X 0,Y 552.2,Z 672.417,A -85,B 0,C 180,E1 -3152.735,E2 -3152.735} C_VEL
LIN {X 0,Y 552.016,Z 681.149,A -85,B 0,C 180,E1 -3154.197,E2 -3154.197} C_VEL
LIN {X 0,Y 551.885,Z 689.335,A -85,B 0,C 180,E1 -3155.846,E2 -3155.846} C_VEL
LIN {X 0,Y 551.812,Z 695.291,A -85,B 0,C 180,E1 -3157.316,E2 -3157.316} C_VEL
LIN {X 0,Y 551.746,Z 700.078,A -85,B 0,C 180,E1 -3158.791,E2 -3158.791} C_VEL
LIN {X 0,Y 551.692,Z 703.829,A -85,B 0,C 180,E1 -3160.272,E2 -3160.272} C_VEL
LIN {X 0,Y 551.671,Z 706.521,A -85,B 0,C 180,E1 -3161.76,E2 -3161.76} C_VEL
LIN {X 0,Y 551.653,Z 708.256,A -85,B 0,C 180,E1 -3163.256,E2 -3163.256} C_VEL
LIN {X 0,Y 551.618,Z 708.946,A -85,B 0,C 180,E1 -3164.762,E2 -3164.762} C_VEL
LIN {X 0,Y 551.628,Z 708.644,A -85,B 0,C 180,E1 -3166.277,E2 -3166.277} C_VEL
LIN {X 0,Y 551.657,Z 707.294,A -85,B 0,C 180,E1 -3167.803,E2 -3167.803} C_VEL
LIN {X 0,Y 551.686,Z 704.528,A -85,B 0,C 180,E1 -3169.49,E2 -3169.49} C_VEL
LIN {X 0,Y 551.722,Z 701.211,A -85,B 0,C 180,E1 -3170.895,E2 -3170.895} C_VEL
LIN {X 0,Y 551.802,Z 696.364,A -85,B 0,C 180,E1 -3172.462,E2 -3172.462} C_VEL
LIN {X 0,Y 551.883,Z 690.196,A -85,B 0,C 180,E1 -3174.047,E2 -3174.047} C_VEL
LIN {X 0,Y 551.962,Z 682.471,A -85,B 0,C 180,E1 -3175.651,E2 -3175.651} C_VEL
LIN {X 0,Y 552.157,Z 674.688,A -85,B 0,C 180,E1 -3177.003,E2 -3177.003} C_VEL
LIN {X 0,Y 552.352,Z 665.576,A -85,B 0,C 180,E1 -3178.347,E2 -3178.347} C_VEL
LIN {X 0,Y 552.607,Z 656.411,A -85,B 0,C 180,E1 -3179.525,E2 -3179.525} C_VEL
LIN {X 0,Y 552.94,Z 645.205,A -85,B 0,C 180,E1 -3180.768,E2 -3180.768} C_VEL
LIN {X 0,Y 553.344,Z 631.464,A -85,B 0,C 180,E1 -3182.066,E2 -3182.066} C_VEL
LIN {X 0,Y 553.732,Z 618.369,A -85,B 0,C 180,E1 -3183.104,E2 -3183.104} C_VEL
LIN {X 0,Y 554.154,Z 605.051,A -85,B 0,C 180,E1 -3184.005,E2 -3184.005} C_VEL
LIN {X 0,Y 554.579,Z 589.652,A -85,B 0,C 180,E1 -3184.878,E2 -3184.878} C_VEL
LIN {X 0,Y 554.903,Z 574.331,A -85,B 0,C 180,E1 -3185.577,E2 -3185.577} C_VEL
LIN {X 0,Y 555.237,Z 559.043,A -85,B 0,C 180,E1 -3186.121,E2 -3186.121} C_VEL
LIN {X 0,Y 555.533,Z 545.111,A -85,B 0,C 180,E1 -3186.501,E2 -3186.501} C_VEL
LIN {X 0,Y 555.567,Z 534.472,A -85,B 0,C 180,E1 -3186.724,E2 -3186.724} C_VEL
LIN {X 0,Y 551.873,Z 521.652,A -85,B 0,C 180,E1 -3187.086,E2 -3187.086} C_VEL
LIN {X 0,Y 551.87,Z 515.743,A -85,B 0,C 180,E1 -3190.173,E2 -3190.173} C_VEL
LIN {X 0,Y 551.952,Z 511.487,A -85,B 0,C 180,E1 -3192.441,E2 -3192.441} C_VEL
LIN {X 0,Y 552.008,Z 505.802,A -85,B 0,C 180,E1 -3195.553,E2 -3195.553} C_VEL
LIN {X 0,Y 552.061,Z 500.549,A -85,B 0,C 180,E1 -3198.548,E2 -3198.548} C_VEL
LIN {X 0,Y 552.075,Z 495.199,A -85,B 0,C 180,E1 -3201.407,E2 -3201.407} C_VEL
LIN {X 0,Y 552.136,Z 490.026,A -85,B 0,C 180,E1 -3204.16,E2 -3204.16} C_VEL
LIN {X 0,Y 552.123,Z 490.025,A -85,B 0,C 180,E1 -3207.15,E2 -3207.15} C_VEL
LIN {X 0,Y 552.138,Z 490.022,A -85,B 0,C 180,E1 -3210.236,E2 -3210.236} C_VEL
LIN {X 0,Y 552.139,Z 490.021,A -85,B 0,C 180,E1 -3212.997,E2 -3212.997} C_VEL
LIN {X 0,Y 552.122,Z 490.025,A -85,B 0,C 180,E1 -3215.161,E2 -3215.161} C_VEL
LIN {X 0,Y 552.107,Z 490.029,A -85,B 0,C 180,E1 -3217.549,E2 -3217.549} C_VEL
LIN {X 0,Y 552.149,Z 490.02,A -85,B 0,C 180,E1 -3220.674,E2 -3220.674} C_VEL
LIN {X 0,Y 552.112,Z 490.023,A -85,B 0,C 180,E1 -3223.737,E2 -3223.737} C_VEL
LIN {X 0,Y 552.129,Z 490.023,A -85,B 0,C 180,E1 -3226.004,E2 -3226.004} C_VEL
LIN {X 0,Y 552.169,Z 490.015,A -85,B 0,C 180,E1 -3228.993,E2 -3228.993} C_VEL
LIN {X 0,Y 552.155,Z 490.017,A -85,B 0,C 180,E1 -3231.951,E2 -3231.951} C_VEL
LIN {X 0,Y 552.23,Z 490.01,A -85,B 0,C 180,E1 -3234.889,E2 -3234.889} C_VEL
LIN {X 0,Y 552.221,Z 490.013,A -85,B 0,C 180,E1 -3237.812,E2 -3237.812} C_VEL
LIN {X 0,Y 552.239,Z 490.011,A -85,B 0,C 180,E1 -3240.729,E2 -3240.729} C_VEL
LIN {X 0,Y 552.202,Z 490.012,A -85,B 0,C 180,E1 -3242.918,E2 -3242.918} C_VEL
LIN {X 0,Y 552.191,Z 490.013,A -85,B 0,C 180,E1 -3245.844,E2 -3245.844} C_VEL
LIN {X 0,Y 552.162,Z 490.019,A -85,B 0,C 180,E1 -3248.785,E2 -3248.785} C_VEL
LIN {X 0,Y 552.153,Z 490.019,A -85,B 0,C 180,E1 -3251.75,E2 -3251.75} C_VEL
LIN {X 0,Y 552.125,Z 490.022,A -85,B 0,C 180,E1 -3254.748,E2 -3254.748} C_VEL
LIN {X 0,Y 552.105,Z 490.015,A -85,B 0,C 180,E1 -3257.788,E2 -3257.788} C_VEL
LIN {X 0,Y 552.124,Z 490.023,A -85,B 0,C 180,E1 -3260.101,E2 -3260.101} C_VEL
LIN {X 0,Y 552.104,Z 490.026,A -85,B 0,C 180,E1 -3262.45,E2 -3262.45} C_VEL
LIN {X 0,Y 552.152,Z 490.017,A -85,B 0,C 180,E1 -3265.353,E2 -3265.353} C_VEL
LIN {X 0,Y 552.117,Z 490.025,A -85,B 0,C 180,E1 -3268.098,E2 -3268.098} C_VEL
LIN {X 0,Y 552.104,Z 490.029,A -85,B 0,C 180,E1 -3270.609,E2 -3270.609} C_VEL
LIN {X 0,Y 552.119,Z 490.026,A -85,B 0,C 180,E1 -3273.185,E2 -3273.185} C_VEL
LIN {X 0,Y 552.105,Z 490.027,A -85,B 0,C 180,E1 -3275.842,E2 -3275.842} C_VEL
LIN {X 0,Y 552.117,Z 490.024,A -85,B 0,C 180,E1 -3279.063,E2 -3279.063} C_VEL
LIN {X 0,Y 552.161,Z 490.021,A -85,B 0,C 180,E1 -3281.442,E2 -3281.442} C_VEL
LIN {X 0,Y 552.087,Z 490.03,A -85,B 0,C 180,E1 -3284.533,E2 -3284.533} C_VEL
LIN {X 0,Y 552.139,Z 490.083,A -85,B 0,C 180,E1 -3287.425,E2 -3287.425} C_VEL
LIN {X 0,Y 554.035,Z 498.634,A -85,B 0,C 180,E1 -3289.69,E2 -3289.69} C_VEL
LIN {X 0,Y 554.312,Z 502.552,A -85,B 0,C 180,E1 -3290.66,E2 -3290.66} C_VEL
LIN {X 0,Y 554.134,Z 511.379,A -85,B 0,C 180,E1 -3292.827,E2 -3292.827} C_VEL
LIN {X 0,Y 553.791,Z 523.604,A -85,B 0,C 180,E1 -3295.813,E2 -3295.813} C_VEL
LIN {X 0,Y 553.504,Z 535.51,A -85,B 0,C 180,E1 -3298.63,E2 -3298.63} C_VEL
LIN {X 0,Y 553.175,Z 548.427,A -85,B 0,C 180,E1 -3301.595,E2 -3301.595} C_VEL
LIN {X 0,Y 552.941,Z 560.938,A -85,B 0,C 180,E1 -3304.397,E2 -3304.397} C_VEL
LIN {X 0,Y 552.641,Z 575.468,A -85,B 0,C 180,E1 -3307.574,E2 -3307.574} C_VEL
LIN {X 0,Y 552.675,Z 577.396,A -85,B 0,C 180,E1 -3307.943,E2 -3307.943} C_VEL
LIN {X 0,Y 555.654,Z 588.657,A -85,B 0,C 180,E1 -3308.226,E2 -3308.226} C_VEL
LIN {X 0,Y 555.523,Z 605.642,A -85,B 0,C 180,E1 -3308.551,E2 -3308.551} C_VEL
LIN {X 0,Y 555.257,Z 622.281,A -85,B 0,C 180,E1 -3309.026,E2 -3309.026} C_VEL
LIN {X 0,Y 554.855,Z 637.512,A -85,B 0,C 180,E1 -3309.604,E2 -3309.604} C_VEL
LIN {X 0,Y 554.46,Z 653.545,A -85,B 0,C 180,E1 -3310.374,E2 -3310.374} C_VEL
LIN {X 0,Y 554.058,Z 668.022,A -85,B 0,C 180,E1 -3311.225,E2 -3311.225} C_VEL
LIN {X 0,Y 553.593,Z 682.718,A -85,B 0,C 180,E1 -3312.262,E2 -3312.262} C_VEL
LIN {X 0,Y 553.189,Z 696.108,A -85,B 0,C 180,E1 -3313.391,E2 -3313.391} C_VEL
LIN {X 0,Y 552.889,Z 707.516,A -85,B 0,C 180,E1 -3314.519,E2 -3314.519} C_VEL
LIN {X 0,Y 552.561,Z 718.943,A -85,B 0,C 180,E1 -3315.829,E2 -3315.829} C_VEL
LIN {X 0,Y 552.276,Z 728.739,A -85,B 0,C 180,E1 -3317.133,E2 -3317.133} C_VEL
LIN {X 0,Y 552.11,Z 738.743,A -85,B 0,C 180,E1 -3318.716,E2 -3318.716} C_VEL
LIN {X 0,Y 551.866,Z 747.861,A -85,B 0,C 180,E1 -3320.471,E2 -3320.471} C_VEL
LIN {X 0,Y 551.804,Z 755.47,A -85,B 0,C 180,E1 -3322.316,E2 -3322.316} C_VEL
LIN {X 0,Y 551.769,Z 761.249,A -85,B 0,C 180,E1 -3324.152,E2 -3324.152} C_VEL
LIN {X 0,Y 551.702,Z 764.637,A -85,B 0,C 180,E1 -3325.617,E2 -3325.617} C_VEL
LIN {X 0,Y 551.712,Z 767.089,A -85,B 0,C 180,E1 -3327.08,E2 -3327.08} C_VEL
LIN {X 0,Y 551.641,Z 768.479,A -85,B 0,C 180,E1 -3328.541,E2 -3328.541} C_VEL
LIN {X 0,Y 551.636,Z 769,A -85,B 0,C 180,E1 -3330.001,E2 -3330.001} C_VEL
LIN {X 0,Y 551.642,Z 768.478,A -85,B 0,C 180,E1 -3331.461,E2 -3331.461} C_VEL
LIN {X 0,Y 551.712,Z 767.087,A -85,B 0,C 180,E1 -3332.921,E2 -3332.921} C_VEL
LIN {X 0,Y 551.702,Z 764.634,A -85,B 0,C 180,E1 -3334.384,E2 -3334.384} C_VEL
LIN {X 0,Y 551.769,Z 761.246,A -85,B 0,C 180,E1 -3335.849,E2 -3335.849} C_VEL
LIN {X 0,Y 551.805,Z 755.466,A -85,B 0,C 180,E1 -3337.686,E2 -3337.686} C_VEL
LIN {X 0,Y 551.867,Z 747.854,A -85,B 0,C 180,E1 -3339.53,E2 -3339.53} C_VEL
LIN {X 0,Y 552.113,Z 738.734,A -85,B 0,C 180,E1 -3341.285,E2 -3341.285} C_VEL
LIN {X 0,Y 552.277,Z 728.729,A -85,B 0,C 180,E1 -3342.868,E2 -3342.868} C_VEL
LIN {X 0,Y 552.627,Z 717.44,A -85,B 0,C 180,E1 -3344.359,E2 -3344.359} C_VEL
LIN {X 0,Y 552.93,Z 705.721,A -85,B 0,C 180,E1 -3345.671,E2 -3345.671} C_VEL
LIN {X 0,Y 553.318,Z 692.911,A -85,B 0,C 180,E1 -3346.891,E2 -3346.891} C_VEL
LIN {X 0,Y 553.728,Z 679.28,A -85,B 0,C 180,E1 -3347.993,E2 -3347.993} C_VEL
LIN {X 0,Y 554.138,Z 665.006,A -85,B 0,C 180,E1 -3348.966,E2 -3348.966} C_VEL
LIN {X 0,Y 554.566,Z 649.977,A -85,B 0,C 180,E1 -3349.817,E2 -3349.817} C_VEL
LIN {X 0,Y 554.945,Z 635.284,A -85,B 0,C 180,E1 -3350.488,E2 -3350.488} C_VEL
LIN {X 0,Y 555.299,Z 619.197,A -85,B 0,C 180,E1 -3351.071,E2 -3351.071} C_VEL
LIN {X 0,Y 555.552,Z 603.458,A -85,B 0,C 180,E1 -3351.499,E2 -3351.499} C_VEL
LIN {X 0,Y 555.584,Z 588.34,A -85,B 0,C 180,E1 -3351.782,E2 -3351.782} C_VEL
LIN {X 0,Y 552.653,Z 577.084,A -85,B 0,C 180,E1 -3352.076,E2 -3352.076} C_VEL
LIN {X 0,Y 552.87,Z 562.937,A -85,B 0,C 180,E1 -3355.163,E2 -3355.163} C_VEL
LIN {X 0,Y 553.166,Z 550.032,A -85,B 0,C 180,E1 -3358.04,E2 -3358.04} C_VEL
LIN {X 0,Y 553.448,Z 537.318,A -85,B 0,C 180,E1 -3360.951,E2 -3360.951} C_VEL
LIN {X 0,Y 553.703,Z 526.422,A -85,B 0,C 180,E1 -3363.514,E2 -3363.514} C_VEL
LIN {X 0,Y 554.022,Z 515.525,A -85,B 0,C 180,E1 -3366.148,E2 -3366.148} C_VEL
LIN {X 0,Y 554.287,Z 505.458,A -85,B 0,C 180,E1 -3368.638,E2 -3368.638} C_VEL
LIN {X 0,Y 553.928,Z 498.5,A -85,B 0,C 180,E1 -3370.083,E2 -3370.083} C_VEL
LIN {X 0,Y 552.156,Z 490.02,A -85,B 0,C 180,E1 -3371.89,E2 -3371.89} C_VEL
LIN {X 0,Y 552.098,Z 490.029,A -85,B 0,C 180,E1 -3374.532,E2 -3374.532} C_VEL
LIN {X 0,Y 552.13,Z 490.019,A -85,B 0,C 180,E1 -3377.585,E2 -3377.585} C_VEL
LIN {X 0,Y 552.135,Z 490.025,A -85,B 0,C 180,E1 -3380.474,E2 -3380.474} C_VEL
LIN {X 0,Y 552.112,Z 490.021,A -85,B 0,C 180,E1 -3383.317,E2 -3383.317} C_VEL
LIN {X 0,Y 552.131,Z 490.022,A -85,B 0,C 180,E1 -3385.94,E2 -3385.94} C_VEL
LIN {X 0,Y 552.12,Z 490.025,A -85,B 0,C 180,E1 -3388.541,E2 -3388.541} C_VEL
LIN {X 0,Y 552.127,Z 490.02,A -85,B 0,C 180,E1 -3391.438,E2 -3391.438} C_VEL
LIN {X 0,Y 552.132,Z 490.023,A -85,B 0,C 180,E1 -3394.356,E2 -3394.356} C_VEL
LIN {X 0,Y 552.112,Z 490.022,A -85,B 0,C 180,E1 -3396.759,E2 -3396.759} C_VEL
LIN {X 0,Y 552.117,Z 490.026,A -85,B 0,C 180,E1 -3398.132,E2 -3398.132} C_VEL
LIN {X 0,Y 553.965,Z 494.933,A -85,B 0,C 180,E1 -3398.303,E2 -3398.303} C_VEL
LIN {X 0,Y 555.607,Z 499.162,A -85,B 0,C 180,E1 -3398.454,E2 -3398.454} C_VEL
LIN {X 0,Y 555.374,Z 515.552,A -85,B 0,C 180,E1 -3398.86,E2 -3398.86} C_VEL
LIN {X 0,Y 555.082,Z 530.718,A -85,B 0,C 180,E1 -3399.374,E2 -3399.374} C_VEL
LIN {X 0,Y 554.7,Z 545.201,A -85,B 0,C 180,E1 -3399.996,E2 -3399.996} C_VEL
LIN {X 0,Y 554.288,Z 559.579,A -85,B 0,C 180,E1 -3400.752,E2 -3400.752} C_VEL
LIN {X 0,Y 553.877,Z 574.691,A -85,B 0,C 180,E1 -3401.716,E2 -3401.716} C_VEL
LIN {X 0,Y 553.425,Z 588.171,A -85,B 0,C 180,E1 -3402.744,E2 -3402.744} C_VEL
LIN {X 0,Y 553.032,Z 601.571,A -85,B 0,C 180,E1 -3403.955,E2 -3403.955} C_VEL
LIN {X 0,Y 552.693,Z 613.899,A -85,B 0,C 180,E1 -3405.267,E2 -3405.267} C_VEL
LIN {X 0,Y 552.387,Z 624.397,A -85,B 0,C 180,E1 -3406.574,E2 -3406.574} C_VEL
LIN {X 0,Y 552.2,Z 634.545,A -85,B 0,C 180,E1 -3408.064,E2 -3408.064} C_VEL
LIN {X 0,Y 552.022,Z 642.064,A -85,B 0,C 180,E1 -3409.362,E2 -3409.362} C_VEL
LIN {X 0,Y 551.891,Z 649.311,A -85,B 0,C 180,E1 -3410.841,E2 -3410.841} C_VEL
LIN {X 0,Y 551.806,Z 655.305,A -85,B 0,C 180,E1 -3412.315,E2 -3412.315} C_VEL
LIN {X 0,Y 551.763,Z 659.159,A -85,B 0,C 180,E1 -3413.471,E2 -3413.471} C_VEL
LIN {X 0,Y 551.698,Z 662.967,A -85,B 0,C 180,E1 -3414.884,E2 -3414.884} C_VEL
LIN {X 0,Y 551.728,Z 665.916,A -85,B 0,C 180,E1 -3416.349,E2 -3416.349} C_VEL
LIN {X 0,Y 551.647,Z 667.862,A -85,B 0,C 180,E1 -3417.81,E2 -3417.81} C_VEL
LIN {X 0,Y 551.64,Z 668.852,A -85,B 0,C 180,E1 -3419.27,E2 -3419.27} C_VEL
LIN {X 0,Y 551.639,Z 668.87,A -85,B 0,C 180,E1 -3420.73,E2 -3420.73} C_VEL
LIN {X 0,Y 551.647,Z 667.957,A -85,B 0,C 180,E1 -3422.191,E2 -3422.191} C_VEL
LIN {X 0,Y 551.731,Z 666.063,A -85,B 0,C 180,E1 -3423.652,E2 -3423.652} C_VEL
LIN {X 0,Y 551.698,Z 663.172,A -85,B 0,C 180,E1 -3425.116,E2 -3425.116} C_VEL
LIN {X 0,Y 551.782,Z 659.218,A -85,B 0,C 180,E1 -3426.6,E2 -3426.6} C_VEL
LIN {X 0,Y 551.827,Z 654.24,A -85,B 0,C 180,E1 -3428.054,E2 -3428.054} C_VEL
LIN {X 0,Y 551.86,Z 648.064,A -85,B 0,C 180,E1 -3429.53,E2 -3429.53} C_VEL
LIN {X 0,Y 552.02,Z 640.529,A -85,B 0,C 180,E1 -3431.01,E2 -3431.01} C_VEL
LIN {X 0,Y 552.212,Z 631.521,A -85,B 0,C 180,E1 -3432.496,E2 -3432.496} C_VEL
LIN {X 0,Y 552.485,Z 620.792,A -85,B 0,C 180,E1 -3433.987,E2 -3433.987} C_VEL
LIN {X 0,Y 552.807,Z 609.846,A -85,B 0,C 180,E1 -3435.28,E2 -3435.28} C_VEL
LIN {X 0,Y 553.197,Z 596.603,A -85,B 0,C 180,E1 -3436.61,E2 -3436.61} C_VEL
LIN {X 0,Y 553.606,Z 582.466,A -85,B 0,C 180,E1 -3437.801,E2 -3437.801} C_VEL
LIN {X 0,Y 554.05,Z 568.699,A -85,B 0,C 180,E1 -3438.777,E2 -3438.777} C_VEL
LIN {X 0,Y 554.441,Z 554.354,A -85,B 0,C 180,E1 -3439.628,E2 -3439.628} C_VEL
LIN {X 0,Y 554.861,Z 538.574,A -85,B 0,C 180,E1 -3440.397,E2 -3440.397} C_VEL
LIN {X 0,Y 555.268,Z 521.335,A -85,B 0,C 180,E1 -3441.048,E2 -3441.048} C_VEL
LIN {X 0,Y 555.493,Z 506.491,A -85,B 0,C 180,E1 -3441.47,E2 -3441.47} C_VEL
LIN {X 0,Y 555.438,Z 498.52,A -85,B 0,C 180,E1 -3441.657,E2 -3441.657} C_VEL
LIN {X 0,Y 552.194,Z 490.541,A -85,B 0,C 180,E1 -3441.931,E2 -3441.931} C_VEL
LIN {X 0,Y 552.134,Z 490.025,A -85,B 0,C 180,E1 -3441.967,E2 -3441.967} C_VEL
LIN {X 0,Y 552.111,Z 490.026,A -85,B 0,C 180,E1 -3444.749,E2 -3444.749} C_VEL
LIN {X 0,Y 551.476,Z 490.109,A -85,B 0,C 180,E1 -3445.358,E2 -3445.358} C_VEL
LIN {X 0,Y 548.624,Z 490.465,A -85,B 0,C 180,E1 -3446.347,E2 -3446.347} C_VEL
LIN {X 0,Y 546.197,Z 490.764,A -85,B 0,C 180,E1 -3447.144,E2 -3447.144} C_VEL
LIN {X 0,Y 545.159,Z 490.891,A -85,B 0,C 180,E1 -3447.759,E2 -3447.759} C_VEL
LIN {X 0,Y 545.078,Z 490.899,A -85,B 0,C 180,E1 -3447.967,E2 -3447.967} C_VEL
LIN {X 0,Y 545.07,Z 490.901,A -85,B 0,C 180,E1 -3451.048,E2 -3451.048} C_VEL
LIN {X 0,Y 545.071,Z 490.901,A -85,B 0,C 180,E1 -3453.672,E2 -3453.672} C_VEL
LIN {X 0,Y 545.059,Z 490.903,A -85,B 0,C 180,E1 -3456.38,E2 -3456.38} C_VEL
LIN {X 0,Y 545.109,Z 490.897,A -85,B 0,C 180,E1 -3459.324,E2 -3459.324} C_VEL
LIN {X 0,Y 545.082,Z 490.901,A -85,B 0,C 180,E1 -3462.103,E2 -3462.103} C_VEL
LIN {X 0,Y 545.042,Z 490.904,A -85,B 0,C 180,E1 -3465.17,E2 -3465.17} C_VEL
LIN {X 0,Y 545.088,Z 490.899,A -85,B 0,C 180,E1 -3467.898,E2 -3467.898} C_VEL
LIN {X 0,Y 545.087,Z 490.899,A -85,B 0,C 180,E1 -3470.818,E2 -3470.818} C_VEL
LIN {X 0,Y 545.047,Z 490.906,A -85,B 0,C 180,E1 -3473.62,E2 -3473.62} C_VEL
LIN {X 0,Y 545.071,Z 490.904,A -85,B 0,C 180,E1 -3476.328,E2 -3476.328} C_VEL
LIN {X 0,Y 545.072,Z 490.906,A -85,B 0,C 180,E1 -3478.952,E2 -3478.952} C_VEL
LIN {X 0,Y 545.107,Z 490.899,A -85,B 0,C 180,E1 -3481.507,E2 -3481.507} C_VEL
LIN {X 0,Y 545.102,Z 490.902,A -85,B 0,C 180,E1 -3484.491,E2 -3484.491} C_VEL
LIN {X 0,Y 545.114,Z 490.989,A -85,B 0,C 180,E1 -3485.902,E2 -3485.902} C_VEL
LIN {X 0,Y 545.037,Z 496.516,A -85,B 0,C 180,E1 -3488.835,E2 -3488.835} C_VEL
LIN {X 0,Y 545.032,Z 500.776,A -85,B 0,C 180,E1 -3491.193,E2 -3491.193} C_VEL
LIN {X 0,Y 544.969,Z 504.967,A -85,B 0,C 180,E1 -3493.517,E2 -3493.517} C_VEL
LIN {X 0,Y 544.971,Z 508.896,A -85,B 0,C 180,E1 -3495.816,E2 -3495.816} C_VEL
LIN {X 0,Y 544.912,Z 514.39,A -85,B 0,C 180,E1 -3498.844,E2 -3498.844} C_VEL
LIN {X 0,Y 544.839,Z 520.013,A -85,B 0,C 180,E1 -3501.842,E2 -3501.842} C_VEL
LIN {X 0,Y 544.814,Z 521.657,A -85,B 0,C 180,E1 -3502.706,E2 -3502.706} C_VEL
LIN {X 0,Y 549.039,Z 536.442,A -85,B 0,C 180,E1 -3503.13,E2 -3503.13} C_VEL
LIN {X 0,Y 548.748,Z 554.912,A -85,B 0,C 180,E1 -3503.575,E2 -3503.575} C_VEL
LIN {X 0,Y 548.377,Z 569.629,A -85,B 0,C 180,E1 -3504.071,E2 -3504.071} C_VEL
LIN {X 0,Y 547.992,Z 583.565,A -85,B 0,C 180,E1 -3504.664,E2 -3504.664} C_VEL
LIN {X 0,Y 547.611,Z 597.668,A -85,B 0,C 180,E1 -3505.399,E2 -3505.399} C_VEL
LIN {X 0,Y 547.083,Z 613.667,A -85,B 0,C 180,E1 -3506.409,E2 -3506.409} C_VEL
LIN {X 0,Y 546.619,Z 626.885,A -85,B 0,C 180,E1 -3507.42,E2 -3507.42} C_VEL
LIN {X 0,Y 546.224,Z 639.265,A -85,B 0,C 180,E1 -3508.525,E2 -3508.525} C_VEL
LIN {X 0,Y 545.812,Z 651.676,A -85,B 0,C 180,E1 -3509.815,E2 -3509.815} C_VEL
LIN {X 0,Y 545.38,Z 663.57,A -85,B 0,C 180,E1 -3511.291,E2 -3511.291} C_VEL
LIN {X 0,Y 545.194,Z 672.481,A -85,B 0,C 180,E1 -3512.585,E2 -3512.585} C_VEL
LIN {X 0,Y 544.943,Z 681.215,A -85,B 0,C 180,E1 -3514.067,E2 -3514.067} C_VEL
LIN {X 0,Y 544.793,Z 688.583,A -85,B 0,C 180,E1 -3515.551,E2 -3515.551} C_VEL
LIN {X 0,Y 544.732,Z 694.659,A -85,B 0,C 180,E1 -3517.039,E2 -3517.039} C_VEL
LIN {X 0,Y 544.668,Z 699.573,A -85,B 0,C 180,E1 -3518.533,E2 -3518.533} C_VEL
LIN {X 0,Y 544.606,Z 702.589,A -85,B 0,C 180,E1 -3519.657,E2 -3519.657} C_VEL
LIN {X 0,Y 544.622,Z 705.836,A -85,B 0,C 180,E1 -3521.264,E2 -3521.264} C_VEL
LIN {X 0,Y 544.565,Z 707.74,A -85,B 0,C 180,E1 -3522.673,E2 -3522.673} C_VEL
LIN {X 0,Y 544.584,Z 708.795,A -85,B 0,C 180,E1 -3524.193,E2 -3524.193} C_VEL
LIN {X 0,Y 544.525,Z 708.846,A -85,B 0,C 180,E1 -3525.725,E2 -3525.725} C_VEL
LIN {X 0,Y 544.575,Z 707.883,A -85,B 0,C 180,E1 -3527.266,E2 -3527.266} C_VEL
LIN {X 0,Y 544.553,Z 705.842,A -85,B 0,C 180,E1 -3528.822,E2 -3528.822} C_VEL
LIN {X 0,Y 544.594,Z 702.691,A -85,B 0,C 180,E1 -3530.391,E2 -3530.391} C_VEL
LIN {X 0,Y 544.68,Z 698.331,A -85,B 0,C 180,E1 -3531.973,E2 -3531.973} C_VEL
LIN {X 0,Y 544.757,Z 692.304,A -85,B 0,C 180,E1 -3533.653,E2 -3533.653} C_VEL
LIN {X 0,Y 544.88,Z 685.468,A -85,B 0,C 180,E1 -3535.19,E2 -3535.19} C_VEL
LIN {X 0,Y 545.054,Z 676.705,A -85,B 0,C 180,E1 -3536.826,E2 -3536.826} C_VEL
LIN {X 0,Y 545.311,Z 667.39,A -85,B 0,C 180,E1 -3538.269,E2 -3538.269} C_VEL
LIN {X 0,Y 545.571,Z 658.006,A -85,B 0,C 180,E1 -3539.519,E2 -3539.519} C_VEL
LIN {X 0,Y 545.909,Z 648.31,A -85,B 0,C 180,E1 -3540.639,E2 -3540.639} C_VEL
LIN {X 0,Y 546.27,Z 637.58,A -85,B 0,C 180,E1 -3541.726,E2 -3541.726} C_VEL
LIN {X 0,Y 546.661,Z 625.57,A -85,B 0,C 180,E1 -3542.78,E2 -3542.78} C_VEL
LIN {X 0,Y 547.179,Z 611.136,A -85,B 0,C 180,E1 -3543.855,E2 -3543.855} C_VEL
LIN {X 0,Y 547.592,Z 596.908,A -85,B 0,C 180,E1 -3544.735,E2 -3544.735} C_VEL
LIN {X 0,Y 548.01,Z 583.784,A -85,B 0,C 180,E1 -3545.415,E2 -3545.415} C_VEL
LIN {X 0,Y 548.343,Z 570.803,A -85,B 0,C 180,E1 -3545.973,E2 -3545.973} C_VEL
LIN {X 0,Y 548.687,Z 557.084,A -85,B 0,C 180,E1 -3546.447,E2 -3546.447} C_VEL
LIN {X 0,Y 548.953,Z 543.321,A -85,B 0,C 180,E1 -3546.815,E2 -3546.815} C_VEL
LIN {X 0,Y 548.878,Z 535.637,A -85,B 0,C 180,E1 -3546.981,E2 -3546.981} C_VEL
LIN {X 0,Y 544.795,Z 521.642,A -85,B 0,C 180,E1 -3547.393,E2 -3547.393} C_VEL
LIN {X 0,Y 544.81,Z 515.898,A -85,B 0,C 180,E1 -3550.439,E2 -3550.439} C_VEL
LIN {X 0,Y 544.869,Z 510.944,A -85,B 0,C 180,E1 -3553.126,E2 -3553.126} C_VEL
LIN {X 0,Y 544.967,Z 505.409,A -85,B 0,C 180,E1 -3556.233,E2 -3556.233} C_VEL
LIN {X 0,Y 545.013,Z 500.854,A -85,B 0,C 180,E1 -3558.879,E2 -3558.879} C_VEL
LIN {X 0,Y 545.026,Z 495.454,A -85,B 0,C 180,E1 -3561.76,E2 -3561.76} C_VEL
LIN {X 0,Y 545.101,Z 490.902,A -85,B 0,C 180,E1 -3564.107,E2 -3564.107} C_VEL
LIN {X 0,Y 545.076,Z 490.903,A -85,B 0,C 180,E1 -3567.212,E2 -3567.212} C_VEL
LIN {X 0,Y 545.094,Z 490.901,A -85,B 0,C 180,E1 -3569.812,E2 -3569.812} C_VEL
LIN {X 0,Y 545.094,Z 490.899,A -85,B 0,C 180,E1 -3572.824,E2 -3572.824} C_VEL
LIN {X 0,Y 545.06,Z 490.903,A -85,B 0,C 180,E1 -3575.631,E2 -3575.631} C_VEL
LIN {X 0,Y 545.072,Z 490.902,A -85,B 0,C 180,E1 -3578.175,E2 -3578.175} C_VEL
LIN {X 0,Y 545.112,Z 490.899,A -85,B 0,C 180,E1 -3580.414,E2 -3580.414} C_VEL
LIN {X 0,Y 545.068,Z 490.901,A -85,B 0,C 180,E1 -3583.521,E2 -3583.521} C_VEL
LIN {X 0,Y 545.087,Z 490.901,A -85,B 0,C 180,E1 -3585.819,E2 -3585.819} C_VEL
LIN {X 0,Y 545.123,Z 490.894,A -85,B 0,C 180,E1 -3588.849,E2 -3588.849} C_VEL
LIN {X 0,Y 545.125,Z 490.892,A -85,B 0,C 180,E1 -3591.847,E2 -3591.847} C_VEL
LIN {X 0,Y 545.205,Z 490.884,A -85,B 0,C 180,E1 -3594.823,E2 -3594.823} C_VEL
LIN {X 0,Y 545.192,Z 490.888,A -85,B 0,C 180,E1 -3597.783,E2 -3597.783} C_VEL
LIN {X 0,Y 545.208,Z 490.887,A -85,B 0,C 180,E1 -3600.738,E2 -3600.738} C_VEL
LIN {X 0,Y 545.168,Z 490.889,A -85,B 0,C 180,E1 -3602.955,E2 -3602.955} C_VEL
LIN {X 0,Y 545.162,Z 490.889,A -85,B 0,C 180,E1 -3605.919,E2 -3605.919} C_VEL
LIN {X 0,Y 545.118,Z 490.896,A -85,B 0,C 180,E1 -3608.9,E2 -3608.9} C_VEL
LIN {X 0,Y 545.125,Z 490.893,A -85,B 0,C 180,E1 -3611.904,E2 -3611.904} C_VEL
LIN {X 0,Y 545.074,Z 490.9,A -85,B 0,C 180,E1 -3614.944,E2 -3614.944} C_VEL
LIN {X 0,Y 545.073,Z 490.891,A -85,B 0,C 180,E1 -3618.026,E2 -3618.026} C_VEL
LIN {X 0,Y 545.089,Z 490.898,A -85,B 0,C 180,E1 -3620.372,E2 -3620.372} C_VEL
LIN {X 0,Y 545.103,Z 490.895,A -85,B 0,C 180,E1 -3623.558,E2 -3623.558} C_VEL
LIN {X 0,Y 545.081,Z 490.896,A -85,B 0,C 180,E1 -3626,E2 -3626} C_VEL
LIN {X 0,Y 545.083,Z 490.9,A -85,B 0,C 180,E1 -3628.75,E2 -3628.75} C_VEL
LIN {X 0,Y 545.068,Z 490.903,A -85,B 0,C 180,E1 -3631.683,E2 -3631.683} C_VEL
LIN {X 0,Y 545.076,Z 490.903,A -85,B 0,C 180,E1 -3634.563,E2 -3634.563} C_VEL
LIN {X 0,Y 545.06,Z 490.906,A -85,B 0,C 180,E1 -3637.302,E2 -3637.302} C_VEL
LIN {X 0,Y 545.086,Z 490.902,A -85,B 0,C 180,E1 -3640.141,E2 -3640.141} C_VEL
LIN {X 0,Y 545.057,Z 490.906,A -85,B 0,C 180,E1 -3642.698,E2 -3642.698} C_VEL
LIN {X 0,Y 545.055,Z 490.906,A -85,B 0,C 180,E1 -3645.168,E2 -3645.168} C_VEL
LIN {X 0,Y 545.096,Z 490.902,A -85,B 0,C 180,E1 -3647.066,E2 -3647.066} C_VEL
LIN {X 0,Y 547.236,Z 500.678,A -85,B 0,C 180,E1 -3649.692,E2 -3649.692} C_VEL
LIN {X 0,Y 547.448,Z 507.33,A -85,B 0,C 180,E1 -3651.334,E2 -3651.334} C_VEL
LIN {X 0,Y 547.178,Z 518.262,A -85,B 0,C 180,E1 -3654.015,E2 -3654.015} C_VEL
LIN {X 0,Y 546.785,Z 530.491,A -85,B 0,C 180,E1 -3656.994,E2 -3656.994} C_VEL
LIN {X 0,Y 546.479,Z 541.09,A -85,B 0,C 180,E1 -3659.502,E2 -3659.502} C_VEL
LIN {X 0,Y 546.205,Z 553.673,A -85,B 0,C 180,E1 -3662.407,E2 -3662.407} C_VEL
LIN {X 0,Y 545.875,Z 566.386,A -85,B 0,C 180,E1 -3665.266,E2 -3665.266} C_VEL
LIN {X 0,Y 545.694,Z 577.336,A -85,B 0,C 180,E1 -3667.644,E2 -3667.644} C_VEL
LIN {X 0,Y 549.111,Z 590.559,A -85,B 0,C 180,E1 -3667.984,E2 -3667.984} C_VEL
LIN {X 0,Y 548.886,Z 606.557,A -85,B 0,C 180,E1 -3668.303,E2 -3668.303} C_VEL
LIN {X 0,Y 548.602,Z 623.033,A -85,B 0,C 180,E1 -3668.784,E2 -3668.784} C_VEL
LIN {X 0,Y 548.152,Z 638.387,A -85,B 0,C 180,E1 -3669.382,E2 -3669.382} C_VEL
LIN {X 0,Y 547.746,Z 653.544,A -85,B 0,C 180,E1 -3670.123,E2 -3670.123} C_VEL
LIN {X 0,Y 547.275,Z 668.021,A -85,B 0,C 180,E1 -3670.983,E2 -3670.983} C_VEL
LIN {X 0,Y 546.754,Z 682.717,A -85,B 0,C 180,E1 -3672.032,E2 -3672.032} C_VEL
LIN {X 0,Y 546.32,Z 696.109,A -85,B 0,C 180,E1 -3673.176,E2 -3673.176} C_VEL
LIN {X 0,Y 545.941,Z 707.516,A -85,B 0,C 180,E1 -3674.317,E2 -3674.317} C_VEL
LIN {X 0,Y 545.608,Z 718.943,A -85,B 0,C 180,E1 -3675.644,E2 -3675.644} C_VEL
LIN {X 0,Y 545.265,Z 728.74,A -85,B 0,C 180,E1 -3676.965,E2 -3676.965} C_VEL
LIN {X 0,Y 545.082,Z 738.294,A -85,B 0,C 180,E1 -3678.493,E2 -3678.493} C_VEL
LIN {X 0,Y 544.87,Z 746.055,A -85,B 0,C 180,E1 -3679.973,E2 -3679.973} C_VEL
LIN {X 0,Y 544.749,Z 752.628,A -85,B 0,C 180,E1 -3681.469,E2 -3681.469} C_VEL
LIN {X 0,Y 544.722,Z 757.959,A -85,B 0,C 180,E1 -3682.96,E2 -3682.96} C_VEL
LIN {X 0,Y 544.685,Z 761.249,A -85,B 0,C 180,E1 -3684.076,E2 -3684.076} C_VEL
LIN {X 0,Y 544.6,Z 764.637,A -85,B 0,C 180,E1 -3685.56,E2 -3685.56} C_VEL
LIN {X 0,Y 544.638,Z 767.09,A -85,B 0,C 180,E1 -3687.042,E2 -3687.042} C_VEL
LIN {X 0,Y 544.542,Z 768.48,A -85,B 0,C 180,E1 -3688.522,E2 -3688.522} C_VEL
LIN {X 0,Y 544.536,Z 769,A -85,B 0,C 180,E1 -3690.001,E2 -3690.001} C_VEL
LIN {X 0,Y 544.542,Z 768.479,A -85,B 0,C 180,E1 -3691.48,E2 -3691.48} C_VEL
LIN {X 0,Y 544.639,Z 767.087,A -85,B 0,C 180,E1 -3692.959,E2 -3692.959} C_VEL
LIN {X 0,Y 544.6,Z 764.634,A -85,B 0,C 180,E1 -3694.442,E2 -3694.442} C_VEL
LIN {X 0,Y 544.685,Z 761.246,A -85,B 0,C 180,E1 -3695.926,E2 -3695.926} C_VEL
LIN {X 0,Y 544.74,Z 755.466,A -85,B 0,C 180,E1 -3697.786,E2 -3697.786} C_VEL
LIN {X 0,Y 544.8,Z 747.854,A -85,B 0,C 180,E1 -3699.655,E2 -3699.655} C_VEL
LIN {X 0,Y 545.017,Z 740.259,A -85,B 0,C 180,E1 -3701.153,E2 -3701.153} C_VEL
LIN {X 0,Y 545.229,Z 731.207,A -85,B 0,C 180,E1 -3702.659,E2 -3702.659} C_VEL
LIN {X 0,Y 545.53,Z 720.419,A -85,B 0,C 180,E1 -3704.169,E2 -3704.169} C_VEL
LIN {X 0,Y 545.927,Z 709.279,A -85,B 0,C 180,E1 -3705.494,E2 -3705.494} C_VEL
LIN {X 0,Y 546.263,Z 697.136,A -85,B 0,C 180,E1 -3706.731,E2 -3706.731} C_VEL
LIN {X 0,Y 546.68,Z 684.539,A -85,B 0,C 180,E1 -3707.82,E2 -3707.82} C_VEL
LIN {X 0,Y 547.158,Z 670.842,A -85,B 0,C 180,E1 -3708.828,E2 -3708.828} C_VEL
LIN {X 0,Y 547.657,Z 655.261,A -85,B 0,C 180,E1 -3709.784,E2 -3709.784} C_VEL
LIN {X 0,Y 548.077,Z 640.519,A -85,B 0,C 180,E1 -3710.528,E2 -3710.528} C_VEL
LIN {X 0,Y 548.561,Z 624.329,A -85,B 0,C 180,E1 -3711.17,E2 -3711.17} C_VEL
LIN {X 0,Y 548.873,Z 608.33,A -85,B 0,C 180,E1 -3711.65,E2 -3711.65} C_VEL
LIN {X 0,Y 549.089,Z 592.948,A -85,B 0,C 180,E1 -3711.978,E2 -3711.978} C_VEL
LIN {X 0,Y 548.848,Z 589.169,A -85,B 0,C 180,E1 -3712.05,E2 -3712.05} C_VEL
LIN {X 0,Y 545.66,Z 577.124,A -85,B 0,C 180,E1 -3712.365,E2 -3712.365} C_VEL
LIN {X 0,Y 545.946,Z 563.282,A -85,B 0,C 180,E1 -3715.427,E2 -3715.427} C_VEL
LIN {X 0,Y 546.223,Z 551.849,A -85,B 0,C 180,E1 -3718.011,E2 -3718.011} C_VEL
LIN {X 0,Y 546.539,Z 539.135,A -85,B 0,C 180,E1 -3720.955,E2 -3720.955} C_VEL
LIN {X 0,Y 546.832,Z 528.237,A -85,B 0,C 180,E1 -3723.549,E2 -3723.549} C_VEL
LIN {X 0,Y 547.209,Z 517.339,A -85,B 0,C 180,E1 -3726.214,E2 -3726.214} C_VEL
LIN {X 0,Y 547.384,Z 509.726,A -85,B 0,C 180,E1 -3728.046,E2 -3728.046} C_VEL
LIN {X 0,Y 547.048,Z 500.407,A -85,B 0,C 180,E1 -3729.968,E2 -3729.968} C_VEL
LIN {X 0,Y 545.095,Z 490.9,A -85,B 0,C 180,E1 -3732.033,E2 -3732.033} C_VEL
LIN {X 0,Y 545.065,Z 490.903,A -85,B 0,C 180,E1 -3735.167,E2 -3735.167} C_VEL
LIN {X 0,Y 545.08,Z 490.898,A -85,B 0,C 180,E1 -3737.898,E2 -3737.898} C_VEL
LIN {X 0,Y 545.085,Z 490.902,A -85,B 0,C 180,E1 -3740.819,E2 -3740.819} C_VEL
LIN {X 0,Y 545.051,Z 490.901,A -85,B 0,C 180,E1 -3743.621,E2 -3743.621} C_VEL
LIN {X 0,Y 545.072,Z 490.905,A -85,B 0,C 180,E1 -3746.329,E2 -3746.329} C_VEL
LIN {X 0,Y 545.067,Z 490.899,A -85,B 0,C 180,E1 -3748.953,E2 -3748.953} C_VEL
LIN {X 0,Y 545.105,Z 490.895,A -85,B 0,C 180,E1 -3751.508,E2 -3751.508} C_VEL
LIN {X 0,Y 545.097,Z 490.898,A -85,B 0,C 180,E1 -3754.491,E2 -3754.491} C_VEL
LIN {X 0,Y 545.046,Z 490.904,A -85,B 0,C 180,E1 -3757.243,E2 -3757.243} C_VEL
LIN {X 0,Y 545.058,Z 490.907,A -85,B 0,C 180,E1 -3757.85,E2 -3757.85} C_VEL
LIN {X 0,Y 546.883,Z 495.74,A -85,B 0,C 180,E1 -3758.023,E2 -3758.023} C_VEL
LIN {X 0,Y 548.996,Z 501.034,A -85,B 0,C 180,E1 -3758.22,E2 -3758.22} C_VEL
LIN {X 0,Y 548.676,Z 517.977,A -85,B 0,C 180,E1 -3758.666,E2 -3758.666} C_VEL
LIN {X 0,Y 548.388,Z 532.762,A -85,B 0,C 180,E1 -3759.192,E2 -3759.192} C_VEL
LIN {X 0,Y 547.952,Z 547.191,A -85,B 0,C 180,E1 -3759.837,E2 -3759.837} C_VEL
LIN {X 0,Y 547.505,Z 561.211,A -85,B 0,C 180,E1 -3760.601,E2 -3760.601} C_VEL
LIN {X 0,Y 547.026,Z 576.134,A -85,B 0,C 180,E1 -3761.586,E2 -3761.586} C_VEL
LIN {X 0,Y 546.529,Z 589.423,A -85,B 0,C 180,E1 -3762.627,E2 -3762.627} C_VEL
LIN {X 0,Y 546.116,Z 601.576,A -85,B 0,C 180,E1 -3763.746,E2 -3763.746} C_VEL
LIN {X 0,Y 545.699,Z 613.907,A -85,B 0,C 180,E1 -3765.074,E2 -3765.074} C_VEL
LIN {X 0,Y 545.39,Z 624.405,A -85,B 0,C 180,E1 -3766.398,E2 -3766.398} C_VEL
LIN {X 0,Y 545.157,Z 634.55,A -85,B 0,C 180,E1 -3767.908,E2 -3767.908} C_VEL
LIN {X 0,Y 544.932,Z 644.01,A -85,B 0,C 180,E1 -3769.598,E2 -3769.598} C_VEL
LIN {X 0,Y 544.795,Z 650.921,A -85,B 0,C 180,E1 -3771.095,E2 -3771.095} C_VEL
LIN {X 0,Y 544.715,Z 656.589,A -85,B 0,C 180,E1 -3772.587,E2 -3772.587} C_VEL
LIN {X 0,Y 544.688,Z 661.118,A -85,B 0,C 180,E1 -3774.076,E2 -3774.076} C_VEL
LIN {X 0,Y 544.6,Z 664.555,A -85,B 0,C 180,E1 -3775.56,E2 -3775.56} C_VEL
LIN {X 0,Y 544.643,Z 667.023,A -85,B 0,C 180,E1 -3777.042,E2 -3777.042} C_VEL
LIN {X 0,Y 544.539,Z 668.47,A -85,B 0,C 180,E1 -3778.521,E2 -3778.521} C_VEL
LIN {X 0,Y 544.538,Z 668.996,A -85,B 0,C 180,E1 -3780,E2 -3780} C_VEL
LIN {X 0,Y 544.539,Z 668.526,A -85,B 0,C 180,E1 -3781.479,E2 -3781.479} C_VEL
LIN {X 0,Y 544.644,Z 667.131,A -85,B 0,C 180,E1 -3782.959,E2 -3782.959} C_VEL
LIN {X 0,Y 544.6,Z 664.735,A -85,B 0,C 180,E1 -3784.441,E2 -3784.441} C_VEL
LIN {X 0,Y 544.689,Z 661.36,A -85,B 0,C 180,E1 -3785.925,E2 -3785.925} C_VEL
LIN {X 0,Y 544.716,Z 656.891,A -85,B 0,C 180,E1 -3787.413,E2 -3787.413} C_VEL
LIN {X 0,Y 544.783,Z 651.306,A -85,B 0,C 180,E1 -3788.906,E2 -3788.906} C_VEL
LIN {X 0,Y 544.924,Z 644.468,A -85,B 0,C 180,E1 -3790.403,E2 -3790.403} C_VEL
LIN {X 0,Y 545.143,Z 635.09,A -85,B 0,C 180,E1 -3792.093,E2 -3792.093} C_VEL
LIN {X 0,Y 545.39,Z 625.025,A -85,B 0,C 180,E1 -3793.602,E2 -3793.602} C_VEL
LIN {X 0,Y 545.725,Z 613.947,A -85,B 0,C 180,E1 -3795.012,E2 -3795.012} C_VEL
LIN {X 0,Y 546.1,Z 602.493,A -85,B 0,C 180,E1 -3796.255,E2 -3796.255} C_VEL
LIN {X 0,Y 546.494,Z 590.497,A -85,B 0,C 180,E1 -3797.372,E2 -3797.372} C_VEL
LIN {X 0,Y 546.975,Z 576.969,A -85,B 0,C 180,E1 -3798.446,E2 -3798.446} C_VEL
LIN {X 0,Y 547.461,Z 562.647,A -85,B 0,C 180,E1 -3799.401,E2 -3799.401} C_VEL
LIN {X 0,Y 547.956,Z 546.995,A -85,B 0,C 180,E1 -3800.261,E2 -3800.261} C_VEL
LIN {X 0,Y 548.35,Z 531.479,A -85,B 0,C 180,E1 -3800.947,E2 -3800.947} C_VEL
LIN {X 0,Y 548.686,Z 517.666,A -85,B 0,C 180,E1 -3801.429,E2 -3801.429} C_VEL
LIN {X 0,Y 548.965,Z 503.587,A -85,B 0,C 180,E1 -3801.808,E2 -3801.808} C_VEL
LIN {X 0,Y 548.783,Z 500.229,A -85,B 0,C 180,E1 -3801.896,E2 -3801.896} C_VEL
LIN {X 0,Y 545.151,Z 491.478,A -85,B 0,C 180,E1 -3802.212,E2 -3802.212} C_VEL
LIN {X 0,Y 545.057,Z 490.905,A -85,B 0,C 180,E1 -3802.242,E2 -3802.242} C_VEL
LIN {X 0,Y 545.121,Z 490.896,A -85,B 0,C 180,E1 -3805.18,E2 -3805.18} C_VEL
LIN {X 0,Y 545.078,Z 490.899,A -85,B 0,C 180,E1 -3807.967,E2 -3807.967} C_VEL
LIN {X 0,Y 544.416,Z 490.985,A -85,B 0,C 180,E1 -3808.583,E2 -3808.583} C_VEL
LIN {X 0,Y 541.544,Z 491.34,A -85,B 0,C 180,E1 -3809.584,E2 -3809.584} C_VEL
LIN {X 0,Y 539.117,Z 491.646,A -85,B 0,C 180,E1 -3810.389,E2 -3810.389} C_VEL
LIN {X 0,Y 538.082,Z 491.772,A -85,B 0,C 180,E1 -3811.012,E2 -3811.012} C_VEL
LIN {X 0,Y 538.003,Z 491.782,A -85,B 0,C 180,E1 -3811.222,E2 -3811.222} C_VEL
LIN {X 0,Y 538.029,Z 491.779,A -85,B 0,C 180,E1 -3814.173,E2 -3814.173} C_VEL
LIN {X 0,Y 538.012,Z 491.781,A -85,B 0,C 180,E1 -3817.171,E2 -3817.171} C_VEL
LIN {X 0,Y 538.03,Z 491.778,A -85,B 0,C 180,E1 -3819.797,E2 -3819.797} C_VEL
LIN {X 0,Y 538.023,Z 491.78,A -85,B 0,C 180,E1 -3822.786,E2 -3822.786} C_VEL
LIN {X 0,Y 538.035,Z 491.78,A -85,B 0,C 180,E1 -3825.925,E2 -3825.925} C_VEL
LIN {X 0,Y 538.057,Z 491.776,A -85,B 0,C 180,E1 -3829.252,E2 -3829.252} C_VEL
LIN {X 0,Y 537.998,Z 491.783,A -85,B 0,C 180,E1 -3832.122,E2 -3832.122} C_VEL
LIN {X 0,Y 538.004,Z 491.783,A -85,B 0,C 180,E1 -3834.916,E2 -3834.916} C_VEL
LIN {X 0,Y 538.025,Z 491.784,A -85,B 0,C 180,E1 -3837.617,E2 -3837.617} C_VEL
LIN {X 0,Y 538.022,Z 491.784,A -85,B 0,C 180,E1 -3840.239,E2 -3840.239} C_VEL
LIN {X 0,Y 538.063,Z 491.775,A -85,B 0,C 180,E1 -3842.796,E2 -3842.796} C_VEL
LIN {X 0,Y 538.085,Z 491.802,A -85,B 0,C 180,E1 -3845.818,E2 -3845.818} C_VEL
LIN {X 0,Y 538.011,Z 496.91,A -85,B 0,C 180,E1 -3848.545,E2 -3848.545} C_VEL
LIN {X 0,Y 537.997,Z 501.274,A -85,B 0,C 180,E1 -3850.938,E2 -3850.938} C_VEL
LIN {X 0,Y 537.924,Z 505.46,A -85,B 0,C 180,E1 -3853.295,E2 -3853.295} C_VEL
LIN {X 0,Y 537.944,Z 509.449,A -85,B 0,C 180,E1 -3855.627,E2 -3855.627} C_VEL
LIN {X 0,Y 537.878,Z 514.794,A -85,B 0,C 180,E1 -3858.697,E2 -3858.697} C_VEL
LIN {X 0,Y 537.757,Z 521.124,A -85,B 0,C 180,E1 -3862.112,E2 -3862.112} C_VEL
LIN {X 0,Y 537.767,Z 521.81,A -85,B 0,C 180,E1 -3862.405,E2 -3862.405} C_VEL
LIN {X 0,Y 542.444,Z 537.879,A -85,B 0,C 180,E1 -3862.875,E2 -3862.875} C_VEL
LIN {X 0,Y 542.119,Z 555.598,A -85,B 0,C 180,E1 -3863.322,E2 -3863.322} C_VEL
LIN {X 0,Y 541.73,Z 569.79,A -85,B 0,C 180,E1 -3863.808,E2 -3863.808} C_VEL
LIN {X 0,Y 541.299,Z 583.765,A -85,B 0,C 180,E1 -3864.411,E2 -3864.411} C_VEL
LIN {X 0,Y 540.907,Z 596.195,A -85,B 0,C 180,E1 -3865.061,E2 -3865.061} C_VEL
LIN {X 0,Y 540.445,Z 609.765,A -85,B 0,C 180,E1 -3865.898,E2 -3865.898} C_VEL
LIN {X 0,Y 539.872,Z 624.799,A -85,B 0,C 180,E1 -3867.014,E2 -3867.014} C_VEL
LIN {X 0,Y 539.366,Z 637.45,A -85,B 0,C 180,E1 -3868.132,E2 -3868.132} C_VEL
LIN {X 0,Y 538.981,Z 648.369,A -85,B 0,C 180,E1 -3869.252,E2 -3869.252} C_VEL
LIN {X 0,Y 538.564,Z 659.454,A -85,B 0,C 180,E1 -3870.56,E2 -3870.56} C_VEL
LIN {X 0,Y 538.219,Z 670.176,A -85,B 0,C 180,E1 -3872.057,E2 -3872.057} C_VEL
LIN {X 0,Y 537.918,Z 679.223,A -85,B 0,C 180,E1 -3873.557,E2 -3873.557} C_VEL
LIN {X 0,Y 537.81,Z 685.968,A -85,B 0,C 180,E1 -3874.872,E2 -3874.872} C_VEL
LIN {X 0,Y 537.661,Z 692.378,A -85,B 0,C 180,E1 -3876.342,E2 -3876.342} C_VEL
LIN {X 0,Y 537.647,Z 697.878,A -85,B 0,C 180,E1 -3877.888,E2 -3877.888} C_VEL
LIN {X 0,Y 537.501,Z 703.062,A -85,B 0,C 180,E1 -3879.786,E2 -3879.786} C_VEL
LIN {X 0,Y 537.54,Z 705.974,A -85,B 0,C 180,E1 -3881.309,E2 -3881.309} C_VEL
LIN {X 0,Y 537.47,Z 707.921,A -85,B 0,C 180,E1 -3882.843,E2 -3882.843} C_VEL
LIN {X 0,Y 537.473,Z 708.917,A -85,B 0,C 180,E1 -3884.618,E2 -3884.618} C_VEL
LIN {X 0,Y 537.424,Z 708.782,A -85,B 0,C 180,E1 -3885.938,E2 -3885.938} C_VEL
LIN {X 0,Y 537.484,Z 707.687,A -85,B 0,C 180,E1 -3887.501,E2 -3887.501} C_VEL
LIN {X 0,Y 537.48,Z 705.529,A -85,B 0,C 180,E1 -3889.079,E2 -3889.079} C_VEL
LIN {X 0,Y 537.552,Z 701.146,A -85,B 0,C 180,E1 -3891.071,E2 -3891.071} C_VEL
LIN {X 0,Y 537.627,Z 696.28,A -85,B 0,C 180,E1 -3892.682,E2 -3892.682} C_VEL
LIN {X 0,Y 537.747,Z 690.1,A -85,B 0,C 180,E1 -3894.309,E2 -3894.309} C_VEL
LIN {X 0,Y 537.937,Z 681.236,A -85,B 0,C 180,E1 -3896.164,E2 -3896.164} C_VEL
LIN {X 0,Y 538.145,Z 672.523,A -85,B 0,C 180,E1 -3897.663,E2 -3897.663} C_VEL
LIN {X 0,Y 538.446,Z 663.333,A -85,B 0,C 180,E1 -3899.012,E2 -3899.012} C_VEL
LIN {X 0,Y 538.818,Z 652.682,A -85,B 0,C 180,E1 -3900.359,E2 -3900.359} C_VEL
LIN {X 0,Y 539.31,Z 639.794,A -85,B 0,C 180,E1 -3901.731,E2 -3901.731} C_VEL
LIN {X 0,Y 539.723,Z 627.84,A -85,B 0,C 180,E1 -3902.82,E2 -3902.82} C_VEL
LIN {X 0,Y 540.182,Z 616.176,A -85,B 0,C 180,E1 -3903.738,E2 -3903.738} C_VEL
LIN {X 0,Y 540.683,Z 602.592,A -85,B 0,C 180,E1 -3904.657,E2 -3904.657} C_VEL
LIN {X 0,Y 541.246,Z 585.811,A -85,B 0,C 180,E1 -3905.582,E2 -3905.582} C_VEL
LIN {X 0,Y 541.651,Z 571.991,A -85,B 0,C 180,E1 -3906.196,E2 -3906.196} C_VEL
LIN {X 0,Y 542.05,Z 558.187,A -85,B 0,C 180,E1 -3906.686,E2 -3906.686} C_VEL
LIN {X 0,Y 542.327,Z 544.714,A -85,B 0,C 180,E1 -3907.059,E2 -3907.059} C_VEL
LIN {X 0,Y 542.279,Z 537.087,A -85,B 0,C 180,E1 -3907.236,E2 -3907.236} C_VEL
LIN {X 0,Y 537.725,Z 521.644,A -85,B 0,C 180,E1 -3907.702,E2 -3907.702} C_VEL
LIN {X 0,Y 537.74,Z 515.888,A -85,B 0,C 180,E1 -3910.803,E2 -3910.803} C_VEL
LIN {X 0,Y 537.816,Z 512.056,A -85,B 0,C 180,E1 -3912.963,E2 -3912.963} C_VEL
LIN {X 0,Y 537.914,Z 506.376,A -85,B 0,C 180,E1 -3916.174,E2 -3916.174} C_VEL
LIN {X 0,Y 537.99,Z 501.066,A -85,B 0,C 180,E1 -3919.258,E2 -3919.258} C_VEL
LIN {X 0,Y 537.983,Z 495.707,A -85,B 0,C 180,E1 -3922.121,E2 -3922.121} C_VEL
LIN {X 0,Y 538.063,Z 491.778,A -85,B 0,C 180,E1 -3924.218,E2 -3924.218} C_VEL
LIN {X 0,Y 538.029,Z 491.784,A -85,B 0,C 180,E1 -3926.727,E2 -3926.727} C_VEL
LIN {X 0,Y 538.03,Z 491.783,A -85,B 0,C 180,E1 -3929.553,E2 -3929.553} C_VEL
LIN {X 0,Y 538.041,Z 491.78,A -85,B 0,C 180,E1 -3931.95,E2 -3931.95} C_VEL
LIN {X 0,Y 538.072,Z 491.774,A -85,B 0,C 180,E1 -3934.467,E2 -3934.467} C_VEL
LIN {X 0,Y 538.037,Z 491.777,A -85,B 0,C 180,E1 -3936.929,E2 -3936.929} C_VEL
LIN {X 0,Y 538.069,Z 491.777,A -85,B 0,C 180,E1 -3940.147,E2 -3940.147} C_VEL
LIN {X 0,Y 538.019,Z 491.78,A -85,B 0,C 180,E1 -3943.298,E2 -3943.298} C_VEL
LIN {X 0,Y 538.055,Z 491.779,A -85,B 0,C 180,E1 -3945.63,E2 -3945.63} C_VEL
LIN {X 0,Y 538.08,Z 491.772,A -85,B 0,C 180,E1 -3948.701,E2 -3948.701} C_VEL
LIN {X 0,Y 538.082,Z 491.77,A -85,B 0,C 180,E1 -3951.739,E2 -3951.739} C_VEL
LIN {X 0,Y 538.181,Z 491.759,A -85,B 0,C 180,E1 -3954.755,E2 -3954.755} C_VEL
LIN {X 0,Y 538.163,Z 491.764,A -85,B 0,C 180,E1 -3957.754,E2 -3957.754} C_VEL
LIN {X 0,Y 538.178,Z 491.762,A -85,B 0,C 180,E1 -3960.748,E2 -3960.748} C_VEL
LIN {X 0,Y 538.134,Z 491.765,A -85,B 0,C 180,E1 -3962.994,E2 -3962.994} C_VEL
LIN {X 0,Y 538.115,Z 491.767,A -85,B 0,C 180,E1 -3965.997,E2 -3965.997} C_VEL
LIN {X 0,Y 538.068,Z 491.774,A -85,B 0,C 180,E1 -3969.017,E2 -3969.017} C_VEL
LIN {X 0,Y 538.073,Z 491.77,A -85,B 0,C 180,E1 -3972.062,E2 -3972.062} C_VEL
LIN {X 0,Y 538.034,Z 491.777,A -85,B 0,C 180,E1 -3975.144,E2 -3975.144} C_VEL
LIN {X 0,Y 538.025,Z 491.769,A -85,B 0,C 180,E1 -3978.27,E2 -3978.27} C_VEL
LIN {X 0,Y 538.032,Z 491.778,A -85,B 0,C 180,E1 -3980.651,E2 -3980.651} C_VEL
LIN {X 0,Y 538.03,Z 491.77,A -85,B 0,C 180,E1 -3983.887,E2 -3983.887} C_VEL
LIN {X 0,Y 538.041,Z 491.775,A -85,B 0,C 180,E1 -3986.366,E2 -3986.366} C_VEL
LIN {X 0,Y 538.045,Z 491.778,A -85,B 0,C 180,E1 -3988.939,E2 -3988.939} C_VEL
LIN {X 0,Y 538.018,Z 491.783,A -85,B 0,C 180,E1 -3991.891,E2 -3991.891} C_VEL
LIN {X 0,Y 538.025,Z 491.782,A -85,B 0,C 180,E1 -3994.622,E2 -3994.622} C_VEL
LIN {X 0,Y 538.016,Z 491.781,A -85,B 0,C 180,E1 -3997.174,E2 -3997.174} C_VEL
LIN {X 0,Y 538.046,Z 491.777,A -85,B 0,C 180,E1 -3999.795,E2 -3999.795} C_VEL
LIN {X 0,Y 538.015,Z 491.783,A -85,B 0,C 180,E1 -4002.786,E2 -4002.786} C_VEL
LIN {X 0,Y 538.022,Z 491.782,A -85,B 0,C 180,E1 -4005.926,E2 -4005.926} C_VEL
LIN {X 0,Y 538.052,Z 491.837,A -85,B 0,C 180,E1 -4006.73,E2 -4006.73} C_VEL
LIN {X 0,Y 540.229,Z 501.709,A -85,B 0,C 180,E1 -4009.425,E2 -4009.425} C_VEL
LIN {X 0,Y 540.604,Z 505.635,A -85,B 0,C 180,E1 -4010.432,E2 -4010.432} C_VEL
LIN {X 0,Y 540.434,Z 515.674,A -85,B 0,C 180,E1 -4012.873,E2 -4012.873} C_VEL
LIN {X 0,Y 540.118,Z 526.428,A -85,B 0,C 180,E1 -4015.528,E2 -4015.528} C_VEL
LIN {X 0,Y 539.722,Z 539.142,A -85,B 0,C 180,E1 -4018.611,E2 -4018.611} C_VEL
LIN {X 0,Y 539.329,Z 551.856,A -85,B 0,C 180,E1 -4021.601,E2 -4021.601} C_VEL
LIN {X 0,Y 538.985,Z 564.57,A -85,B 0,C 180,E1 -4024.515,E2 -4024.515} C_VEL
LIN {X 0,Y 538.678,Z 577.133,A -85,B 0,C 180,E1 -4027.331,E2 -4027.331} C_VEL
LIN {X 0,Y 542.537,Z 591.837,A -85,B 0,C 180,E1 -4027.724,E2 -4027.724} C_VEL
LIN {X 0,Y 542.282,Z 607.957,A -85,B 0,C 180,E1 -4028.063,E2 -4028.063} C_VEL
LIN {X 0,Y 541.979,Z 623.146,A -85,B 0,C 180,E1 -4028.516,E2 -4028.516} C_VEL
LIN {X 0,Y 541.478,Z 639.119,A -85,B 0,C 180,E1 -4029.148,E2 -4029.148} C_VEL
LIN {X 0,Y 541.04,Z 653.542,A -85,B 0,C 180,E1 -4029.866,E2 -4029.866} C_VEL
LIN {X 0,Y 540.527,Z 668.019,A -85,B 0,C 180,E1 -4030.737,E2 -4030.737} C_VEL
LIN {X 0,Y 539.96,Z 682.715,A -85,B 0,C 180,E1 -4031.798,E2 -4031.798} C_VEL
LIN {X 0,Y 539.456,Z 696.111,A -85,B 0,C 180,E1 -4032.956,E2 -4032.956} C_VEL
LIN {X 0,Y 539.016,Z 707.516,A -85,B 0,C 180,E1 -4034.11,E2 -4034.11} C_VEL
LIN {X 0,Y 538.641,Z 719.08,A -85,B 0,C 180,E1 -4035.472,E2 -4035.472} C_VEL
LIN {X 0,Y 538.283,Z 728.741,A -85,B 0,C 180,E1 -4036.793,E2 -4036.793} C_VEL
LIN {X 0,Y 538.033,Z 738.808,A -85,B 0,C 180,E1 -4038.429,E2 -4038.429} C_VEL
LIN {X 0,Y 537.831,Z 746.055,A -85,B 0,C 180,E1 -4039.84,E2 -4039.84} C_VEL
LIN {X 0,Y 537.683,Z 752.628,A -85,B 0,C 180,E1 -4041.356,E2 -4041.356} C_VEL
LIN {X 0,Y 537.639,Z 757.959,A -85,B 0,C 180,E1 -4042.867,E2 -4042.867} C_VEL
LIN {X 0,Y 537.585,Z 761.25,A -85,B 0,C 180,E1 -4043.998,E2 -4043.998} C_VEL
LIN {X 0,Y 537.5,Z 764.638,A -85,B 0,C 180,E1 -4045.501,E2 -4045.501} C_VEL
LIN {X 0,Y 537.539,Z 767.09,A -85,B 0,C 180,E1 -4047.003,E2 -4047.003} C_VEL
LIN {X 0,Y 537.447,Z 768.48,A -85,B 0,C 180,E1 -4048.502,E2 -4048.502} C_VEL
LIN {X 0,Y 537.437,Z 769,A -85,B 0,C 180,E1 -4050.001,E2 -4050.001} C_VEL
LIN {X 0,Y 537.448,Z 768.479,A -85,B 0,C 180,E1 -4051.499,E2 -4051.499} C_VEL
LIN {X 0,Y 537.539,Z 767.087,A -85,B 0,C 180,E1 -4052.999,E2 -4052.999} C_VEL
LIN {X 0,Y 537.5,Z 764.634,A -85,B 0,C 180,E1 -4054.5,E2 -4054.5} C_VEL
LIN {X 0,Y 537.586,Z 761.247,A -85,B 0,C 180,E1 -4056.004,E2 -4056.004} C_VEL
LIN {X 0,Y 537.659,Z 755.465,A -85,B 0,C 180,E1 -4057.889,E2 -4057.889} C_VEL
LIN {X 0,Y 537.729,Z 749.486,A -85,B 0,C 180,E1 -4059.403,E2 -4059.403} C_VEL
LIN {X 0,Y 537.885,Z 742.281,A -85,B 0,C 180,E1 -4060.922,E2 -4060.922} C_VEL
LIN {X 0,Y 538.139,Z 733.669,A -85,B 0,C 180,E1 -4062.445,E2 -4062.445} C_VEL
LIN {X 0,Y 538.437,Z 723.331,A -85,B 0,C 180,E1 -4063.974,E2 -4063.974} C_VEL
LIN {X 0,Y 538.826,Z 712.792,A -85,B 0,C 180,E1 -4065.296,E2 -4065.296} C_VEL
LIN {X 0,Y 539.264,Z 700.064,A -85,B 0,C 180,E1 -4066.662,E2 -4066.662} C_VEL
LIN {X 0,Y 539.777,Z 686.784,A -85,B 0,C 180,E1 -4067.867,E2 -4067.867} C_VEL
LIN {X 0,Y 540.347,Z 672.255,A -85,B 0,C 180,E1 -4068.976,E2 -4068.976} C_VEL
LIN {X 0,Y 540.829,Z 658.707,A -85,B 0,C 180,E1 -4069.846,E2 -4069.846} C_VEL
LIN {X 0,Y 541.325,Z 644.314,A -85,B 0,C 180,E1 -4070.609,E2 -4070.609} C_VEL
LIN {X 0,Y 541.814,Z 628.225,A -85,B 0,C 180,E1 -4071.297,E2 -4071.297} C_VEL
LIN {X 0,Y 542.223,Z 611.625,A -85,B 0,C 180,E1 -4071.839,E2 -4071.839} C_VEL
LIN {X 0,Y 542.452,Z 595.381,A -85,B 0,C 180,E1 -4072.22,E2 -4072.22} C_VEL
LIN {X 0,Y 542.346,Z 590.78,A -85,B 0,C 180,E1 -4072.302,E2 -4072.302} C_VEL
LIN {X 0,Y 538.709,Z 577.066,A -85,B 0,C 180,E1 -4072.682,E2 -4072.682} C_VEL
LIN {X 0,Y 539.089,Z 562.717,A -85,B 0,C 180,E1 -4075.903,E2 -4075.903} C_VEL
LIN {X 0,Y 539.401,Z 550.032,A -85,B 0,C 180,E1 -4078.822,E2 -4078.822} C_VEL
LIN {X 0,Y 539.748,Z 537.461,A -85,B 0,C 180,E1 -4081.792,E2 -4081.792} C_VEL
LIN {X 0,Y 540.206,Z 524.472,A -85,B 0,C 180,E1 -4084.954,E2 -4084.954} C_VEL
LIN {X 0,Y 540.407,Z 517.253,A -85,B 0,C 180,E1 -4086.744,E2 -4086.744} C_VEL
LIN {X 0,Y 540.281,Z 504.699,A -85,B 0,C 180,E1 -4089.357,E2 -4089.357} C_VEL
LIN {X 0,Y 539.489,Z 498.63,A -85,B 0,C 180,E1 -4090.644,E2 -4090.644} C_VEL
LIN {X 0,Y 538.05,Z 491.779,A -85,B 0,C 180,E1 -4092.221,E2 -4092.221} C_VEL
LIN {X 0,Y 538.034,Z 491.78,A -85,B 0,C 180,E1 -4095.141,E2 -4095.141} C_VEL
LIN {X 0,Y 538.035,Z 491.778,A -85,B 0,C 180,E1 -4098.228,E2 -4098.228} C_VEL
LIN {X 0,Y 538.016,Z 491.779,A -85,B 0,C 180,E1 -4101.17,E2 -4101.17} C_VEL
LIN {X 0,Y 538.026,Z 491.78,A -85,B 0,C 180,E1 -4104.085,E2 -4104.085} C_VEL
LIN {X 0,Y 538.032,Z 491.779,A -85,B 0,C 180,E1 -4106.728,E2 -4106.728} C_VEL
LIN {X 0,Y 538.027,Z 491.777,A -85,B 0,C 180,E1 -4109.557,E2 -4109.557} C_VEL
LIN {X 0,Y 538.048,Z 491.779,A -85,B 0,C 180,E1 -4111.951,E2 -4111.951} C_VEL
LIN {X 0,Y 538.073,Z 491.774,A -85,B 0,C 180,E1 -4114.468,E2 -4114.468} C_VEL
LIN {X 0,Y 538.034,Z 491.781,A -85,B 0,C 180,E1 -4117.565,E2 -4117.565} C_VEL
LIN {X 0,Y 539.52,Z 495.968,A -85,B 0,C 180,E1 -4117.711,E2 -4117.711} C_VEL
LIN {X 0,Y 542.307,Z 502.534,A -85,B 0,C 180,E1 -4117.972,E2 -4117.972} C_VEL
LIN {X 0,Y 542.026,Z 519.881,A -85,B 0,C 180,E1 -4118.452,E2 -4118.452} C_VEL
LIN {X 0,Y 541.662,Z 535.04,A -85,B 0,C 180,E1 -4119.017,E2 -4119.017} C_VEL
LIN {X 0,Y 541.095,Z 550.945,A -85,B 0,C 180,E1 -4119.769,E2 -4119.769} C_VEL
LIN {X 0,Y 540.609,Z 565.846,A -85,B 0,C 180,E1 -4120.64,E2 -4120.64} C_VEL
LIN {X 0,Y 540.096,Z 579.627,A -85,B 0,C 180,E1 -4121.606,E2 -4121.606} C_VEL
LIN {X 0,Y 539.589,Z 592.474,A -85,B 0,C 180,E1 -4122.666,E2 -4122.666} C_VEL
LIN {X 0,Y 539.077,Z 605.334,A -85,B 0,C 180,E1 -4123.917,E2 -4123.917} C_VEL
LIN {X 0,Y 538.708,Z 617.352,A -85,B 0,C 180,E1 -4125.296,E2 -4125.296} C_VEL
LIN {X 0,Y 538.28,Z 628.423,A -85,B 0,C 180,E1 -4126.792,E2 -4126.792} C_VEL
LIN {X 0,Y 538.041,Z 638.54,A -85,B 0,C 180,E1 -4128.426,E2 -4128.426} C_VEL
LIN {X 0,Y 537.835,Z 645.866,A -85,B 0,C 180,E1 -4129.84,E2 -4129.84} C_VEL
LIN {X 0,Y 537.688,Z 652.465,A -85,B 0,C 180,E1 -4131.355,E2 -4131.355} C_VEL
LIN {X 0,Y 537.643,Z 657.836,A -85,B 0,C 180,E1 -4132.867,E2 -4132.867} C_VEL
LIN {X 0,Y 537.589,Z 661.118,A -85,B 0,C 180,E1 -4133.997,E2 -4133.997} C_VEL
LIN {X 0,Y 537.501,Z 664.557,A -85,B 0,C 180,E1 -4135.501,E2 -4135.501} C_VEL
LIN {X 0,Y 537.543,Z 667.022,A -85,B 0,C 180,E1 -4137.003,E2 -4137.003} C_VEL
LIN {X 0,Y 537.444,Z 668.473,A -85,B 0,C 180,E1 -4138.502,E2 -4138.502} C_VEL
LIN {X 0,Y 537.439,Z 668.996,A -85,B 0,C 180,E1 -4140,E2 -4140} C_VEL
LIN {X 0,Y 537.445,Z 668.527,A -85,B 0,C 180,E1 -4141.499,E2 -4141.499} C_VEL
LIN {X 0,Y 537.544,Z 667.129,A -85,B 0,C 180,E1 -4142.998,E2 -4142.998} C_VEL
LIN {X 0,Y 537.501,Z 664.736,A -85,B 0,C 180,E1 -4144.5,E2 -4144.5} C_VEL
LIN {X 0,Y 537.59,Z 661.357,A -85,B 0,C 180,E1 -4146.004,E2 -4146.004} C_VEL
LIN {X 0,Y 537.637,Z 656.892,A -85,B 0,C 180,E1 -4147.512,E2 -4147.512} C_VEL
LIN {X 0,Y 537.723,Z 651.304,A -85,B 0,C 180,E1 -4149.024,E2 -4149.024} C_VEL
LIN {X 0,Y 537.873,Z 644.468,A -85,B 0,C 180,E1 -4150.541,E2 -4150.541} C_VEL
LIN {X 0,Y 538.098,Z 636.224,A -85,B 0,C 180,E1 -4152.063,E2 -4152.063} C_VEL
LIN {X 0,Y 538.363,Z 626.379,A -85,B 0,C 180,E1 -4153.591,E2 -4153.591} C_VEL
LIN {X 0,Y 538.711,Z 615.876,A -85,B 0,C 180,E1 -4154.977,E2 -4154.977} C_VEL
LIN {X 0,Y 539.129,Z 604.334,A -85,B 0,C 180,E1 -4156.277,E2 -4156.277} C_VEL
LIN {X 0,Y 539.545,Z 592.347,A -85,B 0,C 180,E1 -4157.434,E2 -4157.434} C_VEL
LIN {X 0,Y 540.115,Z 578.243,A -85,B 0,C 180,E1 -4158.59,E2 -4158.59} C_VEL
LIN {X 0,Y 540.673,Z 564.208,A -85,B 0,C 180,E1 -4159.556,E2 -4159.556} C_VEL
LIN {X 0,Y 541.144,Z 550.808,A -85,B 0,C 180,E1 -4160.329,E2 -4160.329} C_VEL
LIN {X 0,Y 541.647,Z 535.46,A -85,B 0,C 180,E1 -4161.056,E2 -4161.056} C_VEL
LIN {X 0,Y 542.01,Z 519.658,A -85,B 0,C 180,E1 -4161.641,E2 -4161.641} C_VEL
LIN {X 0,Y 542.318,Z 505.832,A -85,B 0,C 180,E1 -4162.032,E2 -4162.032} C_VEL
LIN {X 0,Y 542.114,Z 502.06,A -85,B 0,C 180,E1 -4162.134,E2 -4162.134} C_VEL
LIN {X 0,Y 538.049,Z 492.079,A -85,B 0,C 180,E1 -4162.509,E2 -4162.509} C_VEL
LIN {X 0,Y 538.005,Z 491.783,A -85,B 0,C 180,E1 -4162.565,E2 -4162.565} C_VEL
LIN {X 0,Y 538.048,Z 491.778,A -85,B 0,C 180,E1 -4165.673,E2 -4165.673} C_VEL
LIN {X 0,Y 538.044,Z 491.776,A -85,B 0,C 180,E1 -4168.05,E2 -4168.05} C_VEL
LIN {X 0,Y 538.024,Z 491.781,A -85,B 0,C 180,E1 -4170.627,E2 -4170.627} C_VEL
LIN {X 0,Y 538.003,Z 491.782,A -85,B 0,C 180,E1 -4171.222,E2 -4171.222} C_VEL
LIN {X 0,Y 537.344,Z 491.867,A -85,B 0,C 180,E1 -4171.848,E2 -4171.848} C_VEL
LIN {X 0,Y 534.484,Z 492.221,A -85,B 0,C 180,E1 -4172.862,E2 -4172.862} C_VEL
LIN {X 0,Y 532.074,Z 492.52,A -85,B 0,C 180,E1 -4173.679,E2 -4173.679} C_VEL
LIN {X 0,Y 531.061,Z 492.648,A -85,B 0,C 180,E1 -4174.31,E2 -4174.31} C_VEL
LIN {X 0,Y 530.99,Z 492.657,A -85,B 0,C 180,E1 -4174.524,E2 -4174.524} C_VEL
LIN {X 0,Y 530.971,Z 492.661,A -85,B 0,C 180,E1 -4177.508,E2 -4177.508} C_VEL
LIN {X 0,Y 530.986,Z 492.659,A -85,B 0,C 180,E1 -4180.433,E2 -4180.433} C_VEL
LIN {X 0,Y 530.966,Z 492.661,A -85,B 0,C 180,E1 -4183.281,E2 -4183.281} C_VEL
LIN {X 0,Y 530.987,Z 492.655,A -85,B 0,C 180,E1 -4185.622,E2 -4185.622} C_VEL
LIN {X 0,Y 531.005,Z 492.654,A -85,B 0,C 180,E1 -4188.565,E2 -4188.565} C_VEL
LIN {X 0,Y 530.963,Z 492.66,A -85,B 0,C 180,E1 -4191.529,E2 -4191.529} C_VEL
LIN {X 0,Y 530.96,Z 492.662,A -85,B 0,C 180,E1 -4194.38,E2 -4194.38} C_VEL
LIN {X 0,Y 530.973,Z 492.66,A -85,B 0,C 180,E1 -4197.133,E2 -4197.133} C_VEL
LIN {X 0,Y 530.975,Z 492.659,A -85,B 0,C 180,E1 -4199.803,E2 -4199.803} C_VEL
LIN {X 0,Y 531.019,Z 492.652,A -85,B 0,C 180,E1 -4202.467,E2 -4202.467} C_VEL
LIN {X 0,Y 531.067,Z 492.649,A -85,B 0,C 180,E1 -4205.675,E2 -4205.675} C_VEL
LIN {X 0,Y 530.983,Z 498.824,A -85,B 0,C 180,E1 -4209.061,E2 -4209.061} C_VEL
LIN {X 0,Y 530.949,Z 503.188,A -85,B 0,C 180,E1 -4211.477,E2 -4211.477} C_VEL
LIN {X 0,Y 530.91,Z 508.733,A -85,B 0,C 180,E1 -4214.647,E2 -4214.647} C_VEL
LIN {X 0,Y 530.783,Z 514.087,A -85,B 0,C 180,E1 -4217.768,E2 -4217.768} C_VEL
LIN {X 0,Y 530.681,Z 518.002,A -85,B 0,C 180,E1 -4220.086,E2 -4220.086} C_VEL
LIN {X 0,Y 530.697,Z 521.648,A -85,B 0,C 180,E1 -4222.073,E2 -4222.073} C_VEL
LIN {X 0,Y 535.816,Z 538.746,A -85,B 0,C 180,E1 -4222.603,E2 -4222.603} C_VEL
LIN {X 0,Y 535.506,Z 556.133,A -85,B 0,C 180,E1 -4223.058,E2 -4223.058} C_VEL
LIN {X 0,Y 535.092,Z 570.018,A -85,B 0,C 180,E1 -4223.542,E2 -4223.542} C_VEL
LIN {X 0,Y 534.611,Z 583.969,A -85,B 0,C 180,E1 -4224.152,E2 -4224.152} C_VEL
LIN {X 0,Y 534.128,Z 598.04,A -85,B 0,C 180,E1 -4224.904,E2 -4224.904} C_VEL
